LIN {X 0,Y 259.412,Z 737.757,A -85,B 0,C 180,E1 -19010.279,E2 -19010.279} C_VEL
LIN {X 0,Y 258.208,Z 750.679,A -85,B 0,C 180,E1 -19011.308,E2 -19011.308} C_VEL
LIN {X 0,Y 256.889,Z 762.034,A -85,B 0,C 180,E1 -19012.52,E2 -19012.52} C_VEL
LIN {X 0,Y 255.443,Z 772.557,A -85,B 0,C 180,E1 -19013.942,E2 -19013.942} C_VEL
LIN {X 0,Y 253.814,Z 782.677,A -85,B 0,C 180,E1 -19015.634,E2 -19015.634} C_VEL
LIN {X 0,Y 252.288,Z 792.086,A -85,B 0,C 180,E1 -19017.598,E2 -19017.598} C_VEL
LIN {X 0,Y 250.698,Z 801.193,A -85,B 0,C 180,E1 -19019.969,E2 -19019.969} C_VEL
LIN {X 0,Y 249.415,Z 808.562,A -85,B 0,C 180,E1 -19022.369,E2 -19022.369} C_VEL
LIN {X 0,Y 248.447,Z 814.636,A -85,B 0,C 180,E1 -19024.883,E2 -19024.883} C_VEL
LIN {X 0,Y 247.734,Z 819.375,A -85,B 0,C 180,E1 -19027.409,E2 -19027.409} C_VEL
LIN {X 0,Y 247.173,Z 822.833,A -85,B 0,C 180,E1 -19029.853,E2 -19029.853} C_VEL
LIN {X 0,Y 246.789,Z 825.879,A -85,B 0,C 180,E1 -19033.114,E2 -19033.114} C_VEL
LIN {X 0,Y 246.747,Z 826.996,A -85,B 0,C 180,E1 -19035.402,E2 -19035.402} C_VEL
LIN {X 0,Y 246.905,Z 827.33,A -85,B 0,C 180,E1 -19037.736,E2 -19037.736} C_VEL
LIN {X 0,Y 247.35,Z 826.83,A -85,B 0,C 180,E1 -19040.097,E2 -19040.097} C_VEL
LIN {X 0,Y 248.008,Z 825.441,A -85,B 0,C 180,E1 -19042.508,E2 -19042.508} C_VEL
LIN {X 0,Y 249.202,Z 822.178,A -85,B 0,C 180,E1 -19045.665,E2 -19045.665} C_VEL
LIN {X 0,Y 250.317,Z 819.07,A -85,B 0,C 180,E1 -19047.762,E2 -19047.762} C_VEL
LIN {X 0,Y 252.087,Z 813.878,A -85,B 0,C 180,E1 -19050.417,E2 -19050.417} C_VEL
LIN {X 0,Y 254.053,Z 807.904,A -85,B 0,C 180,E1 -19052.774,E2 -19052.774} C_VEL
LIN {X 0,Y 256.165,Z 801.239,A -85,B 0,C 180,E1 -19054.87,E2 -19054.87} C_VEL
LIN {X 0,Y 258.677,Z 792.614,A -85,B 0,C 180,E1 -19057.05,E2 -19057.05} C_VEL
LIN {X 0,Y 261.487,Z 782.053,A -85,B 0,C 180,E1 -19059.139,E2 -19059.139} C_VEL
LIN {X 0,Y 263.88,Z 771.777,A -85,B 0,C 180,E1 -19060.757,E2 -19060.757} C_VEL
LIN {X 0,Y 265.994,Z 761.633,A -85,B 0,C 180,E1 -19062.019,E2 -19062.019} C_VEL
LIN {X 0,Y 267.994,Z 749.161,A -85,B 0,C 180,E1 -19063.235,E2 -19063.235} C_VEL
LIN {X 0,Y 269.511,Z 735.967,A -85,B 0,C 180,E1 -19064.192,E2 -19064.192} C_VEL
LIN {X 0,Y 270.642,Z 723.077,A -85,B 0,C 180,E1 -19064.783,E2 -19064.783} C_VEL
LIN {X 0,Y 273.912,Z 663.749,A -85,B 0,C 180,E1 -19066.609,E2 -19066.609} C_VEL
LIN {X 0,Y 268.766,Z 652.292,A -85,B 0,C 180,E1 -19068.036,E2 -19068.036} C_VEL
LIN {X 0,Y 263.392,Z 642.224,A -85,B 0,C 180,E1 -19069.562,E2 -19069.562} C_VEL
LIN {X 0,Y 255.899,Z 629.943,A -85,B 0,C 180,E1 -19071.86,E2 -19071.86} C_VEL
LIN {X 0,Y 252.994,Z 625.595,A -85,B 0,C 180,E1 -19072.82,E2 -19072.82} C_VEL
LIN {X 0,Y 250.001,Z 621.447,A -85,B 0,C 180,E1 -19073.848,E2 -19073.848} C_VEL
LIN {X 0,Y 249.794,Z 620.987,A -85,B 0,C 180,E1 -19073.944,E2 -19073.944} C_VEL
LIN {X 0,Y 249.398,Z 619.817,A -85,B 0,C 180,E1 -19074.835,E2 -19074.835} C_VEL
LIN {X 0,Y 248.951,Z 619.475,A -85,B 0,C 180,E1 -19075.705,E2 -19075.705} C_VEL
LIN {X 0,Y 247.095,Z 619.707,A -85,B 0,C 180,E1 -19077.471,E2 -19077.471} C_VEL
LIN {X 0,Y 242.966,Z 620.26,A -85,B 0,C 180,E1 -19081.103,E2 -19081.103} C_VEL
LIN {X 0,Y 242.555,Z 620.265,A -85,B 0,C 180,E1 -19082.049,E2 -19082.049} C_VEL
LIN {X 0,Y 242.429,Z 620.281,A -85,B 0,C 180,E1 -19086.66,E2 -19086.66} C_VEL
LIN {X 0,Y 242.31,Z 620.295,A -85,B 0,C 180,E1 -19090.023,E2 -19090.023} C_VEL
LIN {X 0,Y 242.16,Z 620.316,A -85,B 0,C 180,E1 -19095.142,E2 -19095.142} C_VEL
LIN {X 0,Y 242.069,Z 620.326,A -85,B 0,C 180,E1 -19098.625,E2 -19098.625} C_VEL
LIN {X 0,Y 242.01,Z 620.331,A -85,B 0,C 180,E1 -19102.181,E2 -19102.181} C_VEL
LIN {X 0,Y 242.064,Z 620.322,A -85,B 0,C 180,E1 -19105.839,E2 -19105.839} C_VEL
LIN {X 0,Y 242.005,Z 620.33,A -85,B 0,C 180,E1 -19109.584,E2 -19109.584} C_VEL
LIN {X 0,Y 241.989,Z 620.338,A -85,B 0,C 180,E1 -19113.492,E2 -19113.492} C_VEL
LIN {X 0,Y 242.009,Z 620.332,A -85,B 0,C 180,E1 -19117.579,E2 -19117.579} C_VEL
LIN {X 0,Y 241.997,Z 620.472,A -85,B 0,C 180,E1 -19120.82,E2 -19120.82} C_VEL
LIN {X 0,Y 243.717,Z 626.064,A -85,B 0,C 180,E1 -19124.952,E2 -19124.952} C_VEL
LIN {X 0,Y 245.608,Z 632.24,A -85,B 0,C 180,E1 -19128.843,E2 -19128.843} C_VEL
LIN {X 0,Y 246.3,Z 634.523,A -85,B 0,C 180,E1 -19130.1,E2 -19130.1} C_VEL
LIN {X 0,Y 248.796,Z 639.028,A -85,B 0,C 180,E1 -19131.04,E2 -19131.04} C_VEL
LIN {X 0,Y 250.278,Z 641.401,A -85,B 0,C 180,E1 -19131.566,E2 -19131.566} C_VEL
LIN {X 0,Y 253.661,Z 647.375,A -85,B 0,C 180,E1 -19132.733,E2 -19132.733} C_VEL
LIN {X 0,Y 258.381,Z 656.509,A -85,B 0,C 180,E1 -19134.278,E2 -19134.278} C_VEL
LIN {X 0,Y 263.504,Z 667.81,A -85,B 0,C 180,E1 -19135.875,E2 -19135.875} C_VEL
LIN {X 0,Y 264.479,Z 670.795,A -85,B 0,C 180,E1 -19136.199,E2 -19136.199} C_VEL
LIN {X 0,Y 266.594,Z 687.408,A -85,B 0,C 180,E1 -19137.319,E2 -19137.319} C_VEL
LIN {X 0,Y 267.059,Z 694.958,A -85,B 0,C 180,E1 -19137.724,E2 -19137.724} C_VEL
LIN {X 0,Y 264.07,Z 745.91,A -85,B 0,C 180,E1 -19139.343,E2 -19139.343} C_VEL
LIN {X 0,Y 262.439,Z 760.152,A -85,B 0,C 180,E1 -19140.082,E2 -19140.082} C_VEL
LIN {X 0,Y 260.483,Z 771.827,A -85,B 0,C 180,E1 -19140.946,E2 -19140.946} C_VEL
LIN {X 0,Y 257.997,Z 784.148,A -85,B 0,C 180,E1 -19142.194,E2 -19142.194} C_VEL
LIN {X 0,Y 255.328,Z 795.293,A -85,B 0,C 180,E1 -19143.651,E2 -19143.651} C_VEL
LIN {X 0,Y 252.655,Z 805.45,A -85,B 0,C 180,E1 -19145.34,E2 -19145.34} C_VEL
LIN {X 0,Y 249.936,Z 814.673,A -85,B 0,C 180,E1 -19147.255,E2 -19147.255} C_VEL
LIN {X 0,Y 247.165,Z 823.89,A -85,B 0,C 180,E1 -19149.66,E2 -19149.66} C_VEL
LIN {X 0,Y 244.913,Z 831.116,A -85,B 0,C 180,E1 -19152.033,E2 -19152.033} C_VEL
LIN {X 0,Y 243.367,Z 836.122,A -85,B 0,C 180,E1 -19154.078,E2 -19154.078} C_VEL
LIN {X 0,Y 241.756,Z 841.03,A -85,B 0,C 180,E1 -19156.552,E2 -19156.552} C_VEL
LIN {X 0,Y 240.801,Z 844.831,A -85,B 0,C 180,E1 -19159.065,E2 -19159.065} C_VEL
LIN {X 0,Y 240.187,Z 847.629,A -85,B 0,C 180,E1 -19161.587,E2 -19161.587} C_VEL
LIN {X 0,Y 239.985,Z 848.983,A -85,B 0,C 180,E1 -19163.273,E2 -19163.273} C_VEL
LIN {X 0,Y 239.883,Z 849.917,A -85,B 0,C 180,E1 -19164.958,E2 -19164.958} C_VEL
LIN {X 0,Y 239.923,Z 850.416,A -85,B 0,C 180,E1 -19166.641,E2 -19166.641} C_VEL
LIN {X 0,Y 239.986,Z 850.517,A -85,B 0,C 180,E1 -19168.322,E2 -19168.322} C_VEL
LIN {X 0,Y 240.04,Z 850.216,A -85,B 0,C 180,E1 -19170,E2 -19170} C_VEL
LIN {X 0,Y 240.008,Z 849.483,A -85,B 0,C 180,E1 -19171.678,E2 -19171.678} C_VEL
LIN {X 0,Y 239.972,Z 848.286,A -85,B 0,C 180,E1 -19173.358,E2 -19173.358} C_VEL
LIN {X 0,Y 239.954,Z 846.459,A -85,B 0,C 180,E1 -19175.23,E2 -19175.23} C_VEL
LIN {X 0,Y 240.119,Z 843.345,A -85,B 0,C 180,E1 -19177.568,E2 -19177.568} C_VEL
LIN {X 0,Y 240.537,Z 838.897,A -85,B 0,C 180,E1 -19180.096,E2 -19180.096} C_VEL
LIN {X 0,Y 241.246,Z 833.19,A -85,B 0,C 180,E1 -19182.62,E2 -19182.62} C_VEL
LIN {X 0,Y 242.509,Z 826.029,A -85,B 0,C 180,E1 -19185.119,E2 -19185.119} C_VEL
LIN {X 0,Y 243.903,Z 817.46,A -85,B 0,C 180,E1 -19187.495,E2 -19187.495} C_VEL
LIN {X 0,Y 245.216,Z 809.762,A -85,B 0,C 180,E1 -19189.243,E2 -19189.243} C_VEL
LIN {X 0,Y 247.061,Z 798.798,A -85,B 0,C 180,E1 -19191.265,E2 -19191.265} C_VEL
LIN {X 0,Y 248.915,Z 787.83,A -85,B 0,C 180,E1 -19192.844,E2 -19192.844} C_VEL
LIN {X 0,Y 250.596,Z 775.59,A -85,B 0,C 180,E1 -19194.214,E2 -19194.214} C_VEL
LIN {X 0,Y 252.105,Z 762.896,A -85,B 0,C 180,E1 -19195.268,E2 -19195.268} C_VEL
LIN {X 0,Y 253.179,Z 749.404,A -85,B 0,C 180,E1 -19196.036,E2 -19196.036} C_VEL
LIN {X 0,Y 254.298,Z 723.087,A -85,B 0,C 180,E1 -19196.916,E2 -19196.916} C_VEL
LIN {X 0,Y 255.425,Z 690.334,A -85,B 0,C 180,E1 -19197.95,E2 -19197.95} C_VEL
LIN {X 0,Y 250.396,Z 651.358,A -85,B 0,C 180,E1 -19199.786,E2 -19199.786} C_VEL
LIN {X 0,Y 245.876,Z 638.506,A -85,B 0,C 180,E1 -19200.761,E2 -19200.761} C_VEL
LIN {X 0,Y 243.435,Z 626.587,A -85,B 0,C 180,E1 -19205.267,E2 -19205.267} C_VEL
LIN {X 0,Y 242.027,Z 620.336,A -85,B 0,C 180,E1 -19207.771,E2 -19207.771} C_VEL
LIN {X 0,Y 241.968,Z 620.346,A -85,B 0,C 180,E1 -19211.915,E2 -19211.915} C_VEL
LIN {X 0,Y 241.977,Z 620.345,A -85,B 0,C 180,E1 -19216.559,E2 -19216.559} C_VEL
LIN {X 0,Y 241.987,Z 620.342,A -85,B 0,C 180,E1 -19220.286,E2 -19220.286} C_VEL
LIN {X 0,Y 242.035,Z 620.337,A -85,B 0,C 180,E1 -19224.496,E2 -19224.496} C_VEL
LIN {X 0,Y 241.974,Z 620.343,A -85,B 0,C 180,E1 -19228.479,E2 -19228.479} C_VEL
LIN {X 0,Y 242.004,Z 620.338,A -85,B 0,C 180,E1 -19232.311,E2 -19232.311} C_VEL
LIN {X 0,Y 242.037,Z 620.333,A -85,B 0,C 180,E1 -19236.013,E2 -19236.013} C_VEL
LIN {X 0,Y 242.031,Z 620.334,A -85,B 0,C 180,E1 -19239.607,E2 -19239.607} C_VEL
LIN {X 0,Y 242.16,Z 620.32,A -85,B 0,C 180,E1 -19243.277,E2 -19243.277} C_VEL
LIN {X 0,Y 242.181,Z 620.314,A -85,B 0,C 180,E1 -19248.279,E2 -19248.279} C_VEL
LIN {X 0,Y 242.421,Z 620.284,A -85,B 0,C 180,E1 -19251.665,E2 -19251.665} C_VEL
LIN {X 0,Y 242.255,Z 620.308,A -85,B 0,C 180,E1 -19255.006,E2 -19255.006} C_VEL
LIN {X 0,Y 242.631,Z 620.257,A -85,B 0,C 180,E1 -19258.339,E2 -19258.339} C_VEL
LIN {X 0,Y 242.631,Z 620.254,A -85,B 0,C 180,E1 -19261.659,E2 -19261.659} C_VEL
LIN {X 0,Y 242.423,Z 620.285,A -85,B 0,C 180,E1 -19266.702,E2 -19266.702} C_VEL
LIN {X 0,Y 242.308,Z 620.297,A -85,B 0,C 180,E1 -19270.021,E2 -19270.021} C_VEL
LIN {X 0,Y 242.15,Z 620.313,A -85,B 0,C 180,E1 -19275.141,E2 -19275.141} C_VEL
LIN {X 0,Y 242.064,Z 620.329,A -85,B 0,C 180,E1 -19278.624,E2 -19278.624} C_VEL
LIN {X 0,Y 242.007,Z 620.334,A -85,B 0,C 180,E1 -19282.18,E2 -19282.18} C_VEL
LIN {X 0,Y 242.061,Z 620.322,A -85,B 0,C 180,E1 -19285.838,E2 -19285.838} C_VEL
LIN {X 0,Y 242.001,Z 620.336,A -85,B 0,C 180,E1 -19289.583,E2 -19289.583} C_VEL
LIN {X 0,Y 241.986,Z 620.339,A -85,B 0,C 180,E1 -19293.491,E2 -19293.491} C_VEL
LIN {X 0,Y 242.007,Z 620.329,A -85,B 0,C 180,E1 -19297.578,E2 -19297.578} C_VEL
LIN {X 0,Y 241.979,Z 620.341,A -85,B 0,C 180,E1 -19301.912,E2 -19301.912} C_VEL
LIN {X 0,Y 241.981,Z 620.34,A -85,B 0,C 180,E1 -19306.558,E2 -19306.558} C_VEL
LIN {X 0,Y 241.977,Z 620.335,A -85,B 0,C 180,E1 -19310.286,E2 -19310.286} C_VEL
LIN {X 0,Y 242.032,Z 620.338,A -85,B 0,C 180,E1 -19314.498,E2 -19314.498} C_VEL
LIN {X 0,Y 241.97,Z 620.339,A -85,B 0,C 180,E1 -19318.48,E2 -19318.48} C_VEL
LIN {X 0,Y 241.998,Z 620.339,A -85,B 0,C 180,E1 -19322.312,E2 -19322.312} C_VEL
LIN {X 0,Y 242.053,Z 620.331,A -85,B 0,C 180,E1 -19326.016,E2 -19326.016} C_VEL
LIN {X 0,Y 242.034,Z 620.333,A -85,B 0,C 180,E1 -19329.608,E2 -19329.608} C_VEL
LIN {X 0,Y 242.16,Z 620.318,A -85,B 0,C 180,E1 -19333.278,E2 -19333.278} C_VEL
LIN {X 0,Y 242.184,Z 620.315,A -85,B 0,C 180,E1 -19338.28,E2 -19338.28} C_VEL
LIN {X 0,Y 242.423,Z 620.283,A -85,B 0,C 180,E1 -19341.666,E2 -19341.666} C_VEL
LIN {X 0,Y 242.257,Z 620.307,A -85,B 0,C 180,E1 -19345.007,E2 -19345.007} C_VEL
LIN {X 0,Y 242.634,Z 620.258,A -85,B 0,C 180,E1 -19348.34,E2 -19348.34} C_VEL
LIN {X 0,Y 242.634,Z 620.259,A -85,B 0,C 180,E1 -19351.66,E2 -19351.66} C_VEL
LIN {X 0,Y 242.421,Z 620.287,A -85,B 0,C 180,E1 -19356.659,E2 -19356.659} C_VEL
LIN {X 0,Y 242.264,Z 620.307,A -85,B 0,C 180,E1 -19360.024,E2 -19360.024} C_VEL
LIN {X 0,Y 242.179,Z 620.32,A -85,B 0,C 180,E1 -19364.119,E2 -19364.119} C_VEL
LIN {X 0,Y 243.197,Z 623.213,A -85,B 0,C 180,E1 -19364.353,E2 -19364.353} C_VEL
LIN {X 0,Y 250.975,Z 640.87,A -85,B 0,C 180,E1 -19365.802,E2 -19365.802} C_VEL
LIN {X 0,Y 256.337,Z 655.837,A -85,B 0,C 180,E1 -19366.839,E2 -19366.839} C_VEL
LIN {X 0,Y 253.594,Z 724.318,A -85,B 0,C 180,E1 -19369.008,E2 -19369.008} C_VEL
LIN {X 0,Y 252.699,Z 738.217,A -85,B 0,C 180,E1 -19369.786,E2 -19369.786} C_VEL
LIN {X 0,Y 251.52,Z 750.319,A -85,B 0,C 180,E1 -19370.763,E2 -19370.763} C_VEL
LIN {X 0,Y 249.946,Z 763.385,A -85,B 0,C 180,E1 -19372.202,E2 -19372.202} C_VEL
LIN {X 0,Y 248.319,Z 774.48,A -85,B 0,C 180,E1 -19373.774,E2 -19373.774} C_VEL
LIN {X 0,Y 246.509,Z 785.512,A -85,B 0,C 180,E1 -19375.771,E2 -19375.771} C_VEL
LIN {X 0,Y 244.819,Z 795.48,A -85,B 0,C 180,E1 -19378.037,E2 -19378.037} C_VEL
LIN {X 0,Y 243.527,Z 802.572,A -85,B 0,C 180,E1 -19380.03,E2 -19380.03} C_VEL
LIN {X 0,Y 242.184,Z 810.192,A -85,B 0,C 180,E1 -19382.697,E2 -19382.697} C_VEL
LIN {X 0,Y 241.131,Z 816.741,A -85,B 0,C 180,E1 -19385.655,E2 -19385.655} C_VEL
LIN {X 0,Y 240.498,Z 820.552,A -85,B 0,C 180,E1 -19387.908,E2 -19387.908} C_VEL
LIN {X 0,Y 239.986,Z 823.774,A -85,B 0,C 180,E1 -19390.413,E2 -19390.413} C_VEL
LIN {X 0,Y 239.704,Z 825.962,A -85,B 0,C 180,E1 -19392.864,E2 -19392.864} C_VEL
LIN {X 0,Y 239.65,Z 827.245,A -85,B 0,C 180,E1 -19395.267,E2 -19395.267} C_VEL
LIN {X 0,Y 239.802,Z 827.71,A -85,B 0,C 180,E1 -19397.619,E2 -19397.619} C_VEL
LIN {X 0,Y 240.228,Z 827.369,A -85,B 0,C 180,E1 -19399.939,E2 -19399.939} C_VEL
LIN {X 0,Y 240.817,Z 826.278,A -85,B 0,C 180,E1 -19402.204,E2 -19402.204} C_VEL
LIN {X 0,Y 242.079,Z 823.294,A -85,B 0,C 180,E1 -19405.568,E2 -19405.568} C_VEL
LIN {X 0,Y 243.825,Z 818.733,A -85,B 0,C 180,E1 -19408.747,E2 -19408.747} C_VEL
LIN {X 0,Y 245.899,Z 813.054,A -85,B 0,C 180,E1 -19411.589,E2 -19411.589} C_VEL
LIN {X 0,Y 248.423,Z 805.642,A -85,B 0,C 180,E1 -19414.361,E2 -19414.361} C_VEL
LIN {X 0,Y 250.798,Z 798.49,A -85,B 0,C 180,E1 -19416.465,E2 -19416.465} C_VEL
LIN {X 0,Y 253.583,Z 789.189,A -85,B 0,C 180,E1 -19418.67,E2 -19418.67} C_VEL
LIN {X 0,Y 256.377,Z 778.677,A -85,B 0,C 180,E1 -19420.619,E2 -19420.619} C_VEL
LIN {X 0,Y 258.893,Z 767.889,A -85,B 0,C 180,E1 -19422.2,E2 -19422.2} C_VEL
LIN {X 0,Y 261.273,Z 755.768,A -85,B 0,C 180,E1 -19423.565,E2 -19423.565} C_VEL
LIN {X 0,Y 263.136,Z 743.169,A -85,B 0,C 180,E1 -19424.642,E2 -19424.642} C_VEL
LIN {X 0,Y 264.315,Z 731.972,A -85,B 0,C 180,E1 -19425.345,E2 -19425.345} C_VEL
LIN {X 0,Y 265.338,Z 718.751,A -85,B 0,C 180,E1 -19425.868,E2 -19425.868} C_VEL
LIN {X 0,Y 268.479,Z 666.273,A -85,B 0,C 180,E1 -19427.495,E2 -19427.495} C_VEL
LIN {X 0,Y 263.835,Z 655.832,A -85,B 0,C 180,E1 -19428.859,E2 -19428.859} C_VEL
LIN {X 0,Y 258.895,Z 646.535,A -85,B 0,C 180,E1 -19430.35,E2 -19430.35} C_VEL
LIN {X 0,Y 252.272,Z 635.35,A -85,B 0,C 180,E1 -19432.497,E2 -19432.497} C_VEL
LIN {X 0,Y 248.99,Z 630.59,A -85,B 0,C 180,E1 -19433.63,E2 -19433.63} C_VEL
LIN {X 0,Y 245.83,Z 626.212,A -85,B 0,C 180,E1 -19434.773,E2 -19434.773} C_VEL
LIN {X 0,Y 243.118,Z 622.829,A -85,B 0,C 180,E1 -19435.805,E2 -19435.805} C_VEL
LIN {X 0,Y 242.633,Z 621.629,A -85,B 0,C 180,E1 -19436.056,E2 -19436.056} C_VEL
LIN {X 0,Y 242.455,Z 620.283,A -85,B 0,C 180,E1 -19437.197,E2 -19437.197} C_VEL
LIN {X 0,Y 242.693,Z 620.256,A -85,B 0,C 180,E1 -19440.001,E2 -19440.001} C_VEL
LIN {X 0,Y 242.555,Z 620.265,A -85,B 0,C 180,E1 -19442.049,E2 -19442.049} C_VEL
LIN {X 0,Y 241.713,Z 620.372,A -85,B 0,C 180,E1 -19443.434,E2 -19443.434} C_VEL
LIN {X 0,Y 238.808,Z 620.738,A -85,B 0,C 180,E1 -19445.695,E2 -19445.695} C_VEL
LIN {X 0,Y 236.434,Z 621.032,A -85,B 0,C 180,E1 -19447.537,E2 -19447.537} C_VEL
LIN {X 0,Y 235.407,Z 621.159,A -85,B 0,C 180,E1 -19448.965,E2 -19448.965} C_VEL
LIN {X 0,Y 235.312,Z 621.167,A -85,B 0,C 180,E1 -19449.449,E2 -19449.449} C_VEL
LIN {X 0,Y 235.1,Z 621.197,A -85,B 0,C 180,E1 -19453.837,E2 -19453.837} C_VEL
LIN {X 0,Y 235.065,Z 621.204,A -85,B 0,C 180,E1 -19457.397,E2 -19457.397} C_VEL
LIN {X 0,Y 234.99,Z 621.206,A -85,B 0,C 180,E1 -19462.011,E2 -19462.011} C_VEL
LIN {X 0,Y 234.965,Z 621.209,A -85,B 0,C 180,E1 -19466.659,E2 -19466.659} C_VEL
LIN {X 0,Y 234.921,Z 621.219,A -85,B 0,C 180,E1 -19470.57,E2 -19470.57} C_VEL
LIN {X 0,Y 234.959,Z 621.208,A -85,B 0,C 180,E1 -19474.634,E2 -19474.634} C_VEL
LIN {X 0,Y 235.001,Z 621.287,A -85,B 0,C 180,E1 -19478.358,E2 -19478.358} C_VEL
LIN {X 0,Y 236.76,Z 626.908,A -85,B 0,C 180,E1 -19483.059,E2 -19483.059} C_VEL
LIN {X 0,Y 238.792,Z 633.746,A -85,B 0,C 180,E1 -19487.726,E2 -19487.726} C_VEL
LIN {X 0,Y 241.533,Z 638.403,A -85,B 0,C 180,E1 -19488.894,E2 -19488.894} C_VEL
LIN {X 0,Y 243.004,Z 640.499,A -85,B 0,C 180,E1 -19489.472,E2 -19489.472} C_VEL
LIN {X 0,Y 246.93,Z 647.301,A -85,B 0,C 180,E1 -19490.978,E2 -19490.978} C_VEL
LIN {X 0,Y 249.888,Z 652.716,A -85,B 0,C 180,E1 -19492.061,E2 -19492.061} C_VEL
LIN {X 0,Y 254.084,Z 660.972,A -85,B 0,C 180,E1 -19493.507,E2 -19493.507} C_VEL
LIN {X 0,Y 258.76,Z 671.596,A -85,B 0,C 180,E1 -19495.067,E2 -19495.067} C_VEL
LIN {X 0,Y 259.488,Z 674.129,A -85,B 0,C 180,E1 -19495.337,E2 -19495.337} C_VEL
LIN {X 0,Y 261.522,Z 691.303,A -85,B 0,C 180,E1 -19496.509,E2 -19496.509} C_VEL
LIN {X 0,Y 261.642,Z 696.477,A -85,B 0,C 180,E1 -19496.758,E2 -19496.758} C_VEL
LIN {X 0,Y 258.552,Z 745.528,A -85,B 0,C 180,E1 -19498.354,E2 -19498.354} C_VEL
LIN {X 0,Y 256.886,Z 759.375,A -85,B 0,C 180,E1 -19499.082,E2 -19499.082} C_VEL
LIN {X 0,Y 254.753,Z 771.597,A -85,B 0,C 180,E1 -19499.999,E2 -19499.999} C_VEL
LIN {X 0,Y 252.179,Z 783.881,A -85,B 0,C 180,E1 -19501.267,E2 -19501.267} C_VEL
LIN {X 0,Y 249.375,Z 795.014,A -85,B 0,C 180,E1 -19502.745,E2 -19502.745} C_VEL
LIN {X 0,Y 246.539,Z 805.158,A -85,B 0,C 180,E1 -19504.459,E2 -19504.459} C_VEL
LIN {X 0,Y 243.426,Z 815.185,A -85,B 0,C 180,E1 -19506.611,E2 -19506.611} C_VEL
LIN {X 0,Y 240.552,Z 824.083,A -85,B 0,C 180,E1 -19509.029,E2 -19509.029} C_VEL
LIN {X 0,Y 238.149,Z 831.268,A -85,B 0,C 180,E1 -19511.504,E2 -19511.504} C_VEL
LIN {X 0,Y 236.538,Z 836.205,A -85,B 0,C 180,E1 -19513.605,E2 -19513.605} C_VEL
LIN {X 0,Y 234.827,Z 841.024,A -85,B 0,C 180,E1 -19516.148,E2 -19516.148} C_VEL
LIN {X 0,Y 233.8,Z 844.738,A -85,B 0,C 180,E1 -19518.733,E2 -19518.733} C_VEL
LIN {X 0,Y 233.129,Z 847.449,A -85,B 0,C 180,E1 -19521.331,E2 -19521.331} C_VEL
LIN {X 0,Y 232.91,Z 848.756,A -85,B 0,C 180,E1 -19523.068,E2 -19523.068} C_VEL
LIN {X 0,Y 232.803,Z 849.694,A -85,B 0,C 180,E1 -19525.029,E2 -19525.029} C_VEL
LIN {X 0,Y 232.914,Z 850.149,A -85,B 0,C 180,E1 -19528.271,E2 -19528.271} C_VEL
LIN {X 0,Y 232.967,Z 849.81,A -85,B 0,C 180,E1 -19530,E2 -19530} C_VEL
LIN {X 0,Y 232.937,Z 849.007,A -85,B 0,C 180,E1 -19531.729,E2 -19531.729} C_VEL
LIN {X 0,Y 232.887,Z 847.771,A -85,B 0,C 180,E1 -19533.46,E2 -19533.46} C_VEL
LIN {X 0,Y 232.903,Z 845.082,A -85,B 0,C 180,E1 -19536.062,E2 -19536.062} C_VEL
LIN {X 0,Y 233.177,Z 841.314,A -85,B 0,C 180,E1 -19538.667,E2 -19538.667} C_VEL
LIN {X 0,Y 233.735,Z 836.362,A -85,B 0,C 180,E1 -19541.27,E2 -19541.27} C_VEL
LIN {X 0,Y 234.672,Z 830.083,A -85,B 0,C 180,E1 -19543.862,E2 -19543.862} C_VEL
LIN {X 0,Y 236.043,Z 822.224,A -85,B 0,C 180,E1 -19546.43,E2 -19546.43} C_VEL
LIN {X 0,Y 236.942,Z 816.796,A -85,B 0,C 180,E1 -19547.9,E2 -19547.9} C_VEL
LIN {X 0,Y 238.858,Z 806.46,A -85,B 0,C 180,E1 -19550.225,E2 -19550.225} C_VEL
LIN {X 0,Y 240.464,Z 797.275,A -85,B 0,C 180,E1 -19551.878,E2 -19551.878} C_VEL
LIN {X 0,Y 242.315,Z 785.977,A -85,B 0,C 180,E1 -19553.502,E2 -19553.502} C_VEL
LIN {X 0,Y 243.835,Z 775.346,A -85,B 0,C 180,E1 -19554.703,E2 -19554.703} C_VEL
LIN {X 0,Y 245.37,Z 762.692,A -85,B 0,C 180,E1 -19555.785,E2 -19555.785} C_VEL
LIN {X 0,Y 246.493,Z 749.289,A -85,B 0,C 180,E1 -19556.569,E2 -19556.569} C_VEL
LIN {X 0,Y 247.58,Z 724.665,A -85,B 0,C 180,E1 -19557.421,E2 -19557.421} C_VEL
LIN {X 0,Y 248.733,Z 690.762,A -85,B 0,C 180,E1 -19558.527,E2 -19558.527} C_VEL
LIN {X 0,Y 243.985,Z 653.427,A -85,B 0,C 180,E1 -19560.349,E2 -19560.349} C_VEL
LIN {X 0,Y 238.628,Z 638.243,A -85,B 0,C 180,E1 -19561.518,E2 -19561.518} C_VEL
LIN {X 0,Y 236.148,Z 626.33,A -85,B 0,C 180,E1 -19566.192,E2 -19566.192} C_VEL
LIN {X 0,Y 234.976,Z 621.217,A -85,B 0,C 180,E1 -19568.36,E2 -19568.36} C_VEL
LIN {X 0,Y 234.957,Z 621.219,A -85,B 0,C 180,E1 -19573.468,E2 -19573.468} C_VEL
LIN {X 0,Y 234.952,Z 621.22,A -85,B 0,C 180,E1 -19576.528,E2 -19576.528} C_VEL
LIN {X 0,Y 234.954,Z 621.218,A -85,B 0,C 180,E1 -19581.085,E2 -19581.085} C_VEL
LIN {X 0,Y 234.959,Z 621.217,A -85,B 0,C 180,E1 -19585.366,E2 -19585.366} C_VEL
LIN {X 0,Y 234.967,Z 621.214,A -85,B 0,C 180,E1 -19590.156,E2 -19590.156} C_VEL
LIN {X 0,Y 234.991,Z 621.208,A -85,B 0,C 180,E1 -19593.793,E2 -19593.793} C_VEL
LIN {X 0,Y 234.994,Z 621.215,A -85,B 0,C 180,E1 -19598.967,E2 -19598.967} C_VEL
LIN {X 0,Y 235.092,Z 621.198,A -85,B 0,C 180,E1 -19603.059,E2 -19603.059} C_VEL
LIN {X 0,Y 235.113,Z 621.195,A -85,B 0,C 180,E1 -19607.921,E2 -19607.921} C_VEL
LIN {X 0,Y 235.371,Z 621.161,A -85,B 0,C 180,E1 -19611.413,E2 -19611.413} C_VEL
LIN {X 0,Y 235.397,Z 621.16,A -85,B 0,C 180,E1 -19613.14,E2 -19613.14} C_VEL
LIN {X 0,Y 235.591,Z 621.134,A -85,B 0,C 180,E1 -19618.29,E2 -19618.29} C_VEL
LIN {X 0,Y 235.591,Z 621.13,A -85,B 0,C 180,E1 -19621.709,E2 -19621.709} C_VEL
LIN {X 0,Y 235.397,Z 621.161,A -85,B 0,C 180,E1 -19626.858,E2 -19626.858} C_VEL
LIN {X 0,Y 235.232,Z 621.177,A -85,B 0,C 180,E1 -19630.326,E2 -19630.326} C_VEL
LIN {X 0,Y 235.101,Z 621.193,A -85,B 0,C 180,E1 -19635.606,E2 -19635.606} C_VEL
LIN {X 0,Y 235.001,Z 621.209,A -85,B 0,C 180,E1 -19639.205,E2 -19639.205} C_VEL
LIN {X 0,Y 234.955,Z 621.21,A -85,B 0,C 180,E1 -19642.882,E2 -19642.882} C_VEL
LIN {X 0,Y 234.962,Z 621.206,A -85,B 0,C 180,E1 -19646.657,E2 -19646.657} C_VEL
LIN {X 0,Y 234.917,Z 621.22,A -85,B 0,C 180,E1 -19650.569,E2 -19650.569} C_VEL
LIN {X 0,Y 234.955,Z 621.212,A -85,B 0,C 180,E1 -19654.633,E2 -19654.633} C_VEL
LIN {X 0,Y 234.961,Z 621.207,A -85,B 0,C 180,E1 -19658.952,E2 -19658.952} C_VEL
LIN {X 0,Y 234.96,Z 621.215,A -85,B 0,C 180,E1 -19663.468,E2 -19663.468} C_VEL
LIN {X 0,Y 234.956,Z 621.215,A -85,B 0,C 180,E1 -19666.531,E2 -19666.531} C_VEL
LIN {X 0,Y 234.95,Z 621.213,A -85,B 0,C 180,E1 -19671.086,E2 -19671.086} C_VEL
LIN {X 0,Y 234.956,Z 621.216,A -85,B 0,C 180,E1 -19675.367,E2 -19675.367} C_VEL
LIN {X 0,Y 234.918,Z 621.213,A -85,B 0,C 180,E1 -19679.431,E2 -19679.431} C_VEL
LIN {X 0,Y 234.99,Z 621.212,A -85,B 0,C 180,E1 -19683.794,E2 -19683.794} C_VEL
LIN {X 0,Y 235.008,Z 621.211,A -85,B 0,C 180,E1 -19688.97,E2 -19688.97} C_VEL
LIN {X 0,Y 235.093,Z 621.2,A -85,B 0,C 180,E1 -19693.059,E2 -19693.059} C_VEL
LIN {X 0,Y 235.144,Z 621.191,A -85,B 0,C 180,E1 -19697.924,E2 -19697.924} C_VEL
LIN {X 0,Y 235.373,Z 621.162,A -85,B 0,C 180,E1 -19701.414,E2 -19701.414} C_VEL
LIN {X 0,Y 235.4,Z 621.161,A -85,B 0,C 180,E1 -19703.141,E2 -19703.141} C_VEL
LIN {X 0,Y 235.594,Z 621.135,A -85,B 0,C 180,E1 -19708.291,E2 -19708.291} C_VEL
LIN {X 0,Y 235.594,Z 621.136,A -85,B 0,C 180,E1 -19711.709,E2 -19711.709} C_VEL
LIN {X 0,Y 235.39,Z 621.164,A -85,B 0,C 180,E1 -19716.859,E2 -19716.859} C_VEL
LIN {X 0,Y 235.211,Z 621.185,A -85,B 0,C 180,E1 -19720.327,E2 -19720.327} C_VEL
LIN {X 0,Y 235.161,Z 621.324,A -85,B 0,C 180,E1 -19723.392,E2 -19723.392} C_VEL
LIN {X 0,Y 236.141,Z 624.059,A -85,B 0,C 180,E1 -19723.609,E2 -19723.609} C_VEL
LIN {X 0,Y 244.656,Z 643.104,A -85,B 0,C 180,E1 -19725.244,E2 -19725.244} C_VEL
LIN {X 0,Y 249.8,Z 657.943,A -85,B 0,C 180,E1 -19726.297,E2 -19726.297} C_VEL
LIN {X 0,Y 246.908,Z 724.994,A -85,B 0,C 180,E1 -19728.477,E2 -19728.477} C_VEL
LIN {X 0,Y 245.963,Z 738.863,A -85,B 0,C 180,E1 -19729.279,E2 -19729.279} C_VEL
LIN {X 0,Y 244.642,Z 751.869,A -85,B 0,C 180,E1 -19730.384,E2 -19730.384} C_VEL
LIN {X 0,Y 243.038,Z 764.664,A -85,B 0,C 180,E1 -19731.858,E2 -19731.858} C_VEL
LIN {X 0,Y 241.248,Z 776.1,A -85,B 0,C 180,E1 -19733.567,E2 -19733.567} C_VEL
LIN {X 0,Y 239.627,Z 785.71,A -85,B 0,C 180,E1 -19735.37,E2 -19735.37} C_VEL
LIN {X 0,Y 237.942,Z 795.373,A -85,B 0,C 180,E1 -19737.615,E2 -19737.615} C_VEL
LIN {X 0,Y 236.505,Z 803.084,A -85,B 0,C 180,E1 -19739.832,E2 -19739.832} C_VEL
LIN {X 0,Y 235.146,Z 810.594,A -85,B 0,C 180,E1 -19742.545,E2 -19742.545} C_VEL
LIN {X 0,Y 234.15,Z 816.516,A -85,B 0,C 180,E1 -19745.271,E2 -19745.271} C_VEL
LIN {X 0,Y 233.449,Z 820.627,A -85,B 0,C 180,E1 -19747.702,E2 -19747.702} C_VEL
LIN {X 0,Y 233.066,Z 822.793,A -85,B 0,C 180,E1 -19749.289,E2 -19749.289} C_VEL
LIN {X 0,Y 232.727,Z 825.249,A -85,B 0,C 180,E1 -19751.632,E2 -19751.632} C_VEL
LIN {X 0,Y 232.564,Z 826.959,A -85,B 0,C 180,E1 -19754.03,E2 -19754.03} C_VEL
LIN {X 0,Y 232.607,Z 827.905,A -85,B 0,C 180,E1 -19756.479,E2 -19756.479} C_VEL
LIN {X 0,Y 232.924,Z 828.02,A -85,B 0,C 180,E1 -19758.965,E2 -19758.965} C_VEL
LIN {X 0,Y 233.515,Z 827.27,A -85,B 0,C 180,E1 -19761.489,E2 -19761.489} C_VEL
LIN {X 0,Y 234.344,Z 825.614,A -85,B 0,C 180,E1 -19764.068,E2 -19764.068} C_VEL
LIN {X 0,Y 235.523,Z 822.97,A -85,B 0,C 180,E1 -19766.668,E2 -19766.668} C_VEL
LIN {X 0,Y 237.404,Z 818.392,A -85,B 0,C 180,E1 -19769.785,E2 -19769.785} C_VEL
LIN {X 0,Y 239.478,Z 812.979,A -85,B 0,C 180,E1 -19772.471,E2 -19772.471} C_VEL
LIN {X 0,Y 242.287,Z 805.43,A -85,B 0,C 180,E1 -19775.32,E2 -19775.32} C_VEL
LIN {X 0,Y 244.941,Z 797.696,A -85,B 0,C 180,E1 -19777.601,E2 -19777.601} C_VEL
LIN {X 0,Y 247.772,Z 788.647,A -85,B 0,C 180,E1 -19779.713,E2 -19779.713} C_VEL
LIN {X 0,Y 250.599,Z 778.442,A -85,B 0,C 180,E1 -19781.61,E2 -19781.61} C_VEL
LIN {X 0,Y 252.941,Z 768.831,A -85,B 0,C 180,E1 -19783.039,E2 -19783.039} C_VEL
LIN {X 0,Y 255.382,Z 757.256,A -85,B 0,C 180,E1 -19784.399,E2 -19784.399} C_VEL
LIN {X 0,Y 257.381,Z 744.94,A -85,B 0,C 180,E1 -19785.497,E2 -19785.497} C_VEL
LIN {X 0,Y 258.752,Z 733.037,A -85,B 0,C 180,E1 -19786.283,E2 -19786.283} C_VEL
LIN {X 0,Y 259.848,Z 720.243,A -85,B 0,C 180,E1 -19786.818,E2 -19786.818} C_VEL
LIN {X 0,Y 262.976,Z 668.382,A -85,B 0,C 180,E1 -19788.478,E2 -19788.478} C_VEL
LIN {X 0,Y 258.153,Z 657.637,A -85,B 0,C 180,E1 -19789.992,E2 -19789.992} C_VEL
LIN {X 0,Y 252.825,Z 647.884,A -85,B 0,C 180,E1 -19791.711,E2 -19791.711} C_VEL
LIN {X 0,Y 247.761,Z 639.457,A -85,B 0,C 180,E1 -19793.486,E2 -19793.486} C_VEL
LIN {X 0,Y 245.515,Z 636.084,A -85,B 0,C 180,E1 -19794.3,E2 -19794.3} C_VEL
LIN {X 0,Y 242.439,Z 631.782,A -85,B 0,C 180,E1 -19795.481,E2 -19795.481} C_VEL
LIN {X 0,Y 239.589,Z 627.891,A -85,B 0,C 180,E1 -19796.638,E2 -19796.638} C_VEL
LIN {X 0,Y 236.184,Z 623.303,A -85,B 0,C 180,E1 -19798.136,E2 -19798.136} C_VEL
LIN {X 0,Y 235.829,Z 622.264,A -85,B 0,C 180,E1 -19798.4,E2 -19798.4} C_VEL
LIN {X 0,Y 235.633,Z 621.132,A -85,B 0,C 180,E1 -19799.574,E2 -19799.574} C_VEL
LIN {X 0,Y 235.538,Z 621.14,A -85,B 0,C 180,E1 -19801.965,E2 -19801.965} C_VEL
LIN {X 0,Y 235.4,Z 621.156,A -85,B 0,C 180,E1 -19806.86,E2 -19806.86} C_VEL
LIN {X 0,Y 235.312,Z 621.167,A -85,B 0,C 180,E1 -19809.449,E2 -19809.449} C_VEL
LIN {X 0,Y 234.588,Z 621.263,A -85,B 0,C 180,E1 -19810.876,E2 -19810.876} C_VEL
LIN {X 0,Y 231.637,Z 621.624,A -85,B 0,C 180,E1 -19813.201,E2 -19813.201} C_VEL
LIN {X 0,Y 229.157,Z 621.936,A -85,B 0,C 180,E1 -19815.098,E2 -19815.098} C_VEL
LIN {X 0,Y 228.108,Z 622.064,A -85,B 0,C 180,E1 -19816.572,E2 -19816.572} C_VEL
LIN {X 0,Y 228.03,Z 622.077,A -85,B 0,C 180,E1 -19817.072,E2 -19817.072} C_VEL
LIN {X 0,Y 227.959,Z 622.084,A -85,B 0,C 180,E1 -19821.714,E2 -19821.714} C_VEL
LIN {X 0,Y 227.939,Z 622.084,A -85,B 0,C 180,E1 -19826.604,E2 -19826.604} C_VEL
LIN {X 0,Y 227.895,Z 622.093,A -85,B 0,C 180,E1 -19830.292,E2 -19830.292} C_VEL
LIN {X 0,Y 227.919,Z 622.159,A -85,B 0,C 180,E1 -19835.323,E2 -19835.323} C_VEL
LIN {X 0,Y 229.132,Z 626.081,A -85,B 0,C 180,E1 -19839.341,E2 -19839.341} C_VEL
LIN {X 0,Y 230.541,Z 630.328,A -85,B 0,C 180,E1 -19842.978,E2 -19842.978} C_VEL
LIN {X 0,Y 231.437,Z 633.257,A -85,B 0,C 180,E1 -19844.996,E2 -19844.996} C_VEL
LIN {X 0,Y 234.475,Z 638.104,A -85,B 0,C 180,E1 -19846.497,E2 -19846.497} C_VEL
LIN {X 0,Y 235.997,Z 640.236,A -85,B 0,C 180,E1 -19847.183,E2 -19847.183} C_VEL
LIN {X 0,Y 239.846,Z 646.466,A -85,B 0,C 180,E1 -19848.851,E2 -19848.851} C_VEL
LIN {X 0,Y 243.116,Z 652.202,A -85,B 0,C 180,E1 -19850.179,E2 -19850.179} C_VEL
LIN {X 0,Y 247.603,Z 660.696,A -85,B 0,C 180,E1 -19851.881,E2 -19851.881} C_VEL
LIN {X 0,Y 253.067,Z 672.736,A -85,B 0,C 180,E1 -19853.841,E2 -19853.841} C_VEL
LIN {X 0,Y 254.508,Z 676.721,A -85,B 0,C 180,E1 -19854.364,E2 -19854.364} C_VEL
LIN {X 0,Y 256.237,Z 692.666,A -85,B 0,C 180,E1 -19855.5,E2 -19855.5} C_VEL
LIN {X 0,Y 256.3,Z 698.424,A -85,B 0,C 180,E1 -19855.775,E2 -19855.775} C_VEL
LIN {X 0,Y 253.22,Z 744.963,A -85,B 0,C 180,E1 -19857.309,E2 -19857.309} C_VEL
LIN {X 0,Y 251.478,Z 758.896,A -85,B 0,C 180,E1 -19858.047,E2 -19858.047} C_VEL
LIN {X 0,Y 249.122,Z 771.638,A -85,B 0,C 180,E1 -19859.013,E2 -19859.013} C_VEL
LIN {X 0,Y 246.428,Z 783.783,A -85,B 0,C 180,E1 -19860.296,E2 -19860.296} C_VEL
LIN {X 0,Y 243.511,Z 794.81,A -85,B 0,C 180,E1 -19861.798,E2 -19861.798} C_VEL
LIN {X 0,Y 240.51,Z 804.871,A -85,B 0,C 180,E1 -19863.537,E2 -19863.537} C_VEL
LIN {X 0,Y 237.492,Z 814.061,A -85,B 0,C 180,E1 -19865.526,E2 -19865.526} C_VEL
LIN {X 0,Y 234.395,Z 823.089,A -85,B 0,C 180,E1 -19867.989,E2 -19867.989} C_VEL
LIN {X 0,Y 231.836,Z 830.411,A -85,B 0,C 180,E1 -19870.522,E2 -19870.522} C_VEL
LIN {X 0,Y 229.728,Z 836.312,A -85,B 0,C 180,E1 -19873.105,E2 -19873.105} C_VEL
LIN {X 0,Y 227.918,Z 841.01,A -85,B 0,C 180,E1 -19875.719,E2 -19875.719} C_VEL
LIN {X 0,Y 226.815,Z 844.64,A -85,B 0,C 180,E1 -19878.381,E2 -19878.381} C_VEL
LIN {X 0,Y 226.091,Z 847.277,A -85,B 0,C 180,E1 -19881.059,E2 -19881.059} C_VEL
LIN {X 0,Y 225.832,Z 848.51,A -85,B 0,C 180,E1 -19882.849,E2 -19882.849} C_VEL
LIN {X 0,Y 225.727,Z 849.473,A -85,B 0,C 180,E1 -19885.091,E2 -19885.091} C_VEL
LIN {X 0,Y 225.842,Z 849.779,A -85,B 0,C 180,E1 -19888.217,E2 -19888.217} C_VEL
LIN {X 0,Y 225.896,Z 849.376,A -85,B 0,C 180,E1 -19890,E2 -19890} C_VEL
LIN {X 0,Y 225.867,Z 848.523,A -85,B 0,C 180,E1 -19891.783,E2 -19891.783} C_VEL
LIN {X 0,Y 225.808,Z 847.25,A -85,B 0,C 180,E1 -19893.569,E2 -19893.569} C_VEL
LIN {X 0,Y 225.832,Z 844.483,A -85,B 0,C 180,E1 -19896.253,E2 -19896.253} C_VEL
LIN {X 0,Y 226.13,Z 840.632,A -85,B 0,C 180,E1 -19898.94,E2 -19898.94} C_VEL
LIN {X 0,Y 226.716,Z 835.585,A -85,B 0,C 180,E1 -19901.624,E2 -19901.624} C_VEL
LIN {X 0,Y 227.763,Z 829.208,A -85,B 0,C 180,E1 -19904.291,E2 -19904.291} C_VEL
LIN {X 0,Y 229.213,Z 821.171,A -85,B 0,C 180,E1 -19906.934,E2 -19906.934} C_VEL
LIN {X 0,Y 230.352,Z 814.135,A -85,B 0,C 180,E1 -19908.838,E2 -19908.838} C_VEL
LIN {X 0,Y 232.295,Z 803.996,A -85,B 0,C 180,E1 -19911.055,E2 -19911.055} C_VEL
LIN {X 0,Y 234.274,Z 793.083,A -85,B 0,C 180,E1 -19912.953,E2 -19912.953} C_VEL
LIN {X 0,Y 236.013,Z 782.46,A -85,B 0,C 180,E1 -19914.404,E2 -19914.404} C_VEL
LIN {X 0,Y 237.781,Z 769.814,A -85,B 0,C 180,E1 -19915.728,E2 -19915.728} C_VEL
LIN {X 0,Y 239.277,Z 756.571,A -85,B 0,C 180,E1 -19916.727,E2 -19916.727} C_VEL
LIN {X 0,Y 240.143,Z 743.256,A -85,B 0,C 180,E1 -19917.388,E2 -19917.388} C_VEL
LIN {X 0,Y 242.2,Z 692.177,A -85,B 0,C 180,E1 -19919.088,E2 -19919.088} C_VEL
LIN {X 0,Y 237.616,Z 655.538,A -85,B 0,C 180,E1 -19920.935,E2 -19920.935} C_VEL
LIN {X 0,Y 231.29,Z 637.905,A -85,B 0,C 180,E1 -19922.341,E2 -19922.341} C_VEL
LIN {X 0,Y 229.3,Z 628.158,A -85,B 0,C 180,E1 -19926.288,E2 -19926.288} C_VEL
LIN {X 0,Y 227.934,Z 622.094,A -85,B 0,C 180,E1 -19928.876,E2 -19928.876} C_VEL
LIN {X 0,Y 227.9,Z 622.101,A -85,B 0,C 180,E1 -19932.72,E2 -19932.72} C_VEL
LIN {X 0,Y 227.893,Z 622.097,A -85,B 0,C 180,E1 -19937.741,E2 -19937.741} C_VEL
LIN {X 0,Y 227.87,Z 622.099,A -85,B 0,C 180,E1 -19941.913,E2 -19941.913} C_VEL
LIN {X 0,Y 227.889,Z 622.098,A -85,B 0,C 180,E1 -19946.372,E2 -19946.372} C_VEL
LIN {X 0,Y 227.917,Z 622.093,A -85,B 0,C 180,E1 -19950.437,E2 -19950.437} C_VEL
LIN {X 0,Y 227.922,Z 622.089,A -85,B 0,C 180,E1 -19954.424,E2 -19954.424} C_VEL
LIN {X 0,Y 227.944,Z 622.091,A -85,B 0,C 180,E1 -19958.284,E2 -19958.284} C_VEL
LIN {X 0,Y 228.031,Z 622.076,A -85,B 0,C 180,E1 -19962.825,E2 -19962.825} C_VEL
LIN {X 0,Y 228.069,Z 622.074,A -85,B 0,C 180,E1 -19967.542,E2 -19967.542} C_VEL
LIN {X 0,Y 228.3,Z 622.039,A -85,B 0,C 180,E1 -19971.145,E2 -19971.145} C_VEL
LIN {X 0,Y 228.349,Z 622.037,A -85,B 0,C 180,E1 -19972.927,E2 -19972.927} C_VEL
LIN {X 0,Y 228.55,Z 622.011,A -85,B 0,C 180,E1 -19978.237,E2 -19978.237} C_VEL
LIN {X 0,Y 228.55,Z 622.007,A -85,B 0,C 180,E1 -19981.761,E2 -19981.761} C_VEL
LIN {X 0,Y 228.348,Z 622.04,A -85,B 0,C 180,E1 -19987.071,E2 -19987.071} C_VEL
LIN {X 0,Y 228.153,Z 622.058,A -85,B 0,C 180,E1 -19990.65,E2 -19990.65} C_VEL
LIN {X 0,Y 228.054,Z 622.068,A -85,B 0,C 180,E1 -19994.272,E2 -19994.272} C_VEL
LIN {X 0,Y 227.997,Z 622.084,A -85,B 0,C 180,E1 -19997.953,E2 -19997.953} C_VEL
LIN {X 0,Y 227.924,Z 622.087,A -85,B 0,C 180,E1 -20002.328,E2 -20002.328} C_VEL
LIN {X 0,Y 227.936,Z 622.081,A -85,B 0,C 180,E1 -20006.602,E2 -20006.602} C_VEL
LIN {X 0,Y 227.891,Z 622.097,A -85,B 0,C 180,E1 -20010.291,E2 -20010.291} C_VEL
LIN {X 0,Y 227.885,Z 622.097,A -85,B 0,C 180,E1 -20013.718,E2 -20013.718} C_VEL
LIN {X 0,Y 227.866,Z 622.089,A -85,B 0,C 180,E1 -20018.086,E2 -20018.086} C_VEL
LIN {X 0,Y 227.904,Z 622.095,A -85,B 0,C 180,E1 -20022.719,E2 -20022.719} C_VEL
LIN {X 0,Y 227.892,Z 622.092,A -85,B 0,C 180,E1 -20027.742,E2 -20027.742} C_VEL
LIN {X 0,Y 227.866,Z 622.096,A -85,B 0,C 180,E1 -20031.914,E2 -20031.914} C_VEL
LIN {X 0,Y 227.886,Z 622.099,A -85,B 0,C 180,E1 -20036.373,E2 -20036.373} C_VEL
LIN {X 0,Y 227.9,Z 622.09,A -85,B 0,C 180,E1 -20040.436,E2 -20040.436} C_VEL
LIN {X 0,Y 227.924,Z 622.095,A -85,B 0,C 180,E1 -20044.426,E2 -20044.426} C_VEL
LIN {X 0,Y 227.959,Z 622.089,A -85,B 0,C 180,E1 -20048.287,E2 -20048.287} C_VEL
LIN {X 0,Y 228.031,Z 622.08,A -85,B 0,C 180,E1 -20052.826,E2 -20052.826} C_VEL
LIN {X 0,Y 228.091,Z 622.07,A -85,B 0,C 180,E1 -20057.545,E2 -20057.545} C_VEL
LIN {X 0,Y 228.302,Z 622.044,A -85,B 0,C 180,E1 -20061.146,E2 -20061.146} C_VEL
LIN {X 0,Y 228.351,Z 622.039,A -85,B 0,C 180,E1 -20062.929,E2 -20062.929} C_VEL
LIN {X 0,Y 228.552,Z 622.012,A -85,B 0,C 180,E1 -20068.238,E2 -20068.238} C_VEL
LIN {X 0,Y 228.552,Z 622.013,A -85,B 0,C 180,E1 -20071.762,E2 -20071.762} C_VEL
LIN {X 0,Y 228.336,Z 622.044,A -85,B 0,C 180,E1 -20077.072,E2 -20077.072} C_VEL
LIN {X 0,Y 228.143,Z 622.067,A -85,B 0,C 180,E1 -20080.651,E2 -20080.651} C_VEL
LIN {X 0,Y 228.096,Z 622.276,A -85,B 0,C 180,E1 -20082.608,E2 -20082.608} C_VEL
LIN {X 0,Y 230.042,Z 627.033,A -85,B 0,C 180,E1 -20083.029,E2 -20083.029} C_VEL
LIN {X 0,Y 238.462,Z 645.693,A -85,B 0,C 180,E1 -20084.698,E2 -20084.698} C_VEL
LIN {X 0,Y 243.186,Z 659.183,A -85,B 0,C 180,E1 -20085.688,E2 -20085.688} C_VEL
LIN {X 0,Y 240.281,Z 725.016,A -85,B 0,C 180,E1 -20087.885,E2 -20087.885} C_VEL
LIN {X 0,Y 239.305,Z 738.957,A -85,B 0,C 180,E1 -20088.708,E2 -20088.708} C_VEL
LIN {X 0,Y 237.999,Z 751.605,A -85,B 0,C 180,E1 -20089.798,E2 -20089.798} C_VEL
LIN {X 0,Y 236.292,Z 764.766,A -85,B 0,C 180,E1 -20091.342,E2 -20091.342} C_VEL
LIN {X 0,Y 234.618,Z 775.224,A -85,B 0,C 180,E1 -20092.918,E2 -20092.918} C_VEL
LIN {X 0,Y 232.701,Z 786.292,A -85,B 0,C 180,E1 -20095.037,E2 -20095.037} C_VEL
LIN {X 0,Y 231.085,Z 795.126,A -85,B 0,C 180,E1 -20097.141,E2 -20097.141} C_VEL
LIN {X 0,Y 229.429,Z 803.695,A -85,B 0,C 180,E1 -20099.666,E2 -20099.666} C_VEL
LIN {X 0,Y 228.012,Z 811.294,A -85,B 0,C 180,E1 -20102.524,E2 -20102.524} C_VEL
LIN {X 0,Y 226.979,Z 817.436,A -85,B 0,C 180,E1 -20105.489,E2 -20105.489} C_VEL
LIN {X 0,Y 226.159,Z 822.007,A -85,B 0,C 180,E1 -20108.425,E2 -20108.425} C_VEL
LIN {X 0,Y 225.628,Z 825.491,A -85,B 0,C 180,E1 -20111.621,E2 -20111.621} C_VEL
LIN {X 0,Y 225.46,Z 827.304,A -85,B 0,C 180,E1 -20114.198,E2 -20114.198} C_VEL
LIN {X 0,Y 225.526,Z 828.262,A -85,B 0,C 180,E1 -20116.72,E2 -20116.72} C_VEL
LIN {X 0,Y 225.87,Z 828.389,A -85,B 0,C 180,E1 -20119.201,E2 -20119.201} C_VEL
LIN {X 0,Y 226.456,Z 827.75,A -85,B 0,C 180,E1 -20121.634,E2 -20121.634} C_VEL
LIN {X 0,Y 227.234,Z 826.413,A -85,B 0,C 180,E1 -20124.011,E2 -20124.011} C_VEL
LIN {X 0,Y 228.862,Z 823.058,A -85,B 0,C 180,E1 -20127.494,E2 -20127.494} C_VEL
LIN {X 0,Y 230.382,Z 819.651,A -85,B 0,C 180,E1 -20129.914,E2 -20129.914} C_VEL
LIN {X 0,Y 232.256,Z 815.176,A -85,B 0,C 180,E1 -20132.365,E2 -20132.365} C_VEL
LIN {X 0,Y 234.966,Z 808.368,A -85,B 0,C 180,E1 -20135.245,E2 -20135.245} C_VEL
LIN {X 0,Y 238.075,Z 800.104,A -85,B 0,C 180,E1 -20137.891,E2 -20137.891} C_VEL
LIN {X 0,Y 241.162,Z 790.948,A -85,B 0,C 180,E1 -20140.208,E2 -20140.208} C_VEL
LIN {X 0,Y 244.158,Z 781.016,A -85,B 0,C 180,E1 -20142.188,E2 -20142.188} C_VEL
LIN {X 0,Y 247.079,Z 769.915,A -85,B 0,C 180,E1 -20143.922,E2 -20143.922} C_VEL
LIN {X 0,Y 249.699,Z 758.3,A -85,B 0,C 180,E1 -20145.327,E2 -20145.327} C_VEL
LIN {X 0,Y 251.838,Z 745.81,A -85,B 0,C 180,E1 -20146.472,E2 -20146.472} C_VEL
LIN {X 0,Y 253.318,Z 733.656,A -85,B 0,C 180,E1 -20147.294,E2 -20147.294} C_VEL
LIN {X 0,Y 254.496,Z 720.657,A -85,B 0,C 180,E1 -20147.846,E2 -20147.846} C_VEL
LIN {X 0,Y 257.707,Z 670.776,A -85,B 0,C 180,E1 -20149.47,E2 -20149.47} C_VEL
LIN {X 0,Y 252.632,Z 659.706,A -85,B 0,C 180,E1 -20151.169,E2 -20151.169} C_VEL
LIN {X 0,Y 246.603,Z 648.801,A -85,B 0,C 180,E1 -20153.295,E2 -20153.295} C_VEL
LIN {X 0,Y 242.313,Z 641.845,A -85,B 0,C 180,E1 -20154.921,E2 -20154.921} C_VEL
LIN {X 0,Y 238.994,Z 637.12,A -85,B 0,C 180,E1 -20156.26,E2 -20156.26} C_VEL
LIN {X 0,Y 236.266,Z 633.201,A -85,B 0,C 180,E1 -20157.444,E2 -20157.444} C_VEL
LIN {X 0,Y 233.257,Z 629.142,A -85,B 0,C 180,E1 -20158.838,E2 -20158.838} C_VEL
LIN {X 0,Y 232.138,Z 627.542,A -85,B 0,C 180,E1 -20159.396,E2 -20159.396} C_VEL
LIN {X 0,Y 229.493,Z 624.691,A -85,B 0,C 180,E1 -20160.714,E2 -20160.714} C_VEL
LIN {X 0,Y 228.774,Z 623.079,A -85,B 0,C 180,E1 -20161.211,E2 -20161.211} C_VEL
LIN {X 0,Y 228.365,Z 622.04,A -85,B 0,C 180,E1 -20162.647,E2 -20162.647} C_VEL
LIN {X 0,Y 228.351,Z 622.035,A -85,B 0,C 180,E1 -20167.072,E2 -20167.072} C_VEL
LIN {X 0,Y 228.155,Z 622.061,A -85,B 0,C 180,E1 -20170.652,E2 -20170.652} C_VEL
LIN {X 0,Y 228.059,Z 622.078,A -85,B 0,C 180,E1 -20174.273,E2 -20174.273} C_VEL
LIN {X 0,Y 228.03,Z 622.077,A -85,B 0,C 180,E1 -20177.072,E2 -20177.072} C_VEL
LIN {X 0,Y 227.369,Z 622.17,A -85,B 0,C 180,E1 -20178.545,E2 -20178.545} C_VEL
LIN {X 0,Y 224.481,Z 622.535,A -85,B 0,C 180,E1 -20180.947,E2 -20180.947} C_VEL
LIN {X 0,Y 222.009,Z 622.836,A -85,B 0,C 180,E1 -20182.907,E2 -20182.907} C_VEL
LIN {X 0,Y 220.938,Z 622.961,A -85,B 0,C 180,E1 -20184.43,E2 -20184.43} C_VEL
LIN {X 0,Y 220.846,Z 622.968,A -85,B 0,C 180,E1 -20184.947,E2 -20184.947} C_VEL
LIN {X 0,Y 220.825,Z 622.967,A -85,B 0,C 180,E1 -20188.516,E2 -20188.516} C_VEL
LIN {X 0,Y 220.845,Z 623.135,A -85,B 0,C 180,E1 -20191.406,E2 -20191.406} C_VEL
LIN {X 0,Y 221.723,Z 625.51,A -85,B 0,C 180,E1 -20194.79,E2 -20194.79} C_VEL
LIN {X 0,Y 222.962,Z 629.463,A -85,B 0,C 180,E1 -20199.082,E2 -20199.082} C_VEL
LIN {X 0,Y 223.901,Z 632.331,A -85,B 0,C 180,E1 -20201.537,E2 -20201.537} C_VEL
LIN {X 0,Y 227.502,Z 637.84,A -85,B 0,C 180,E1 -20203.695,E2 -20203.695} C_VEL
LIN {X 0,Y 228.74,Z 639.465,A -85,B 0,C 180,E1 -20204.347,E2 -20204.347} C_VEL
LIN {X 0,Y 233.005,Z 646.106,A -85,B 0,C 180,E1 -20206.502,E2 -20206.502} C_VEL
LIN {X 0,Y 236.524,Z 651.976,A -85,B 0,C 180,E1 -20208.112,E2 -20208.112} C_VEL
LIN {X 0,Y 239.772,Z 657.921,A -85,B 0,C 180,E1 -20209.514,E2 -20209.514} C_VEL
LIN {X 0,Y 243.534,Z 665.223,A -85,B 0,C 180,E1 -20211.022,E2 -20211.022} C_VEL
LIN {X 0,Y 248.56,Z 676.654,A -85,B 0,C 180,E1 -20212.96,E2 -20212.96} C_VEL
LIN {X 0,Y 249.654,Z 679.718,A -85,B 0,C 180,E1 -20213.378,E2 -20213.378} C_VEL
LIN {X 0,Y 251.178,Z 694.788,A -85,B 0,C 180,E1 -20214.475,E2 -20214.475} C_VEL
LIN {X 0,Y 251.07,Z 700.313,A -85,B 0,C 180,E1 -20214.719,E2 -20214.719} C_VEL
LIN {X 0,Y 247.945,Z 744.559,A -85,B 0,C 180,E1 -20216.213,E2 -20216.213} C_VEL
LIN {X 0,Y 246.133,Z 758.461,A -85,B 0,C 180,E1 -20216.964,E2 -20216.964} C_VEL
LIN {X 0,Y 243.771,Z 770.721,A -85,B 0,C 180,E1 -20217.89,E2 -20217.89} C_VEL
LIN {X 0,Y 240.762,Z 783.745,A -85,B 0,C 180,E1 -20219.281,E2 -20219.281} C_VEL
LIN {X 0,Y 237.701,Z 794.721,A -85,B 0,C 180,E1 -20220.802,E2 -20220.802} C_VEL
LIN {X 0,Y 234.22,Z 805.693,A -85,B 0,C 180,E1 -20222.769,E2 -20222.769} C_VEL
LIN {X 0,Y 231.092,Z 814.657,A -85,B 0,C 180,E1 -20224.801,E2 -20224.801} C_VEL
LIN {X 0,Y 227.836,Z 823.486,A -85,B 0,C 180,E1 -20227.321,E2 -20227.321} C_VEL
LIN {X 0,Y 225.164,Z 830.625,A -85,B 0,C 180,E1 -20229.92,E2 -20229.92} C_VEL
LIN {X 0,Y 222.938,Z 836.404,A -85,B 0,C 180,E1 -20232.574,E2 -20232.574} C_VEL
LIN {X 0,Y 221.03,Z 841.001,A -85,B 0,C 180,E1 -20235.264,E2 -20235.264} C_VEL
LIN {X 0,Y 219.823,Z 844.534,A -85,B 0,C 180,E1 -20238.006,E2 -20238.006} C_VEL
LIN {X 0,Y 219.047,Z 847.092,A -85,B 0,C 180,E1 -20240.769,E2 -20240.769} C_VEL
LIN {X 0,Y 218.648,Z 849.032,A -85,B 0,C 180,E1 -20244.467,E2 -20244.467} C_VEL
LIN {X 0,Y 218.633,Z 849.416,A -85,B 0,C 180,E1 -20246.314,E2 -20246.314} C_VEL
LIN {X 0,Y 218.771,Z 849.397,A -85,B 0,C 180,E1 -20248.159,E2 -20248.159} C_VEL
LIN {X 0,Y 218.826,Z 848.922,A -85,B 0,C 180,E1 -20250,E2 -20250} C_VEL
LIN {X 0,Y 218.798,Z 848.028,A -85,B 0,C 180,E1 -20251.841,E2 -20251.841} C_VEL
LIN {X 0,Y 218.726,Z 845.416,A -85,B 0,C 180,E1 -20255.067,E2 -20255.067} C_VEL
LIN {X 0,Y 218.959,Z 841.357,A -85,B 0,C 180,E1 -20258.305,E2 -20258.305} C_VEL
LIN {X 0,Y 219.483,Z 836.608,A -85,B 0,C 180,E1 -20261.076,E2 -20261.076} C_VEL
LIN {X 0,Y 220.606,Z 829.409,A -85,B 0,C 180,E1 -20264.294,E2 -20264.294} C_VEL
LIN {X 0,Y 222.066,Z 821.551,A -85,B 0,C 180,E1 -20267.022,E2 -20267.022} C_VEL
LIN {X 0,Y 223.004,Z 815.849,A -85,B 0,C 180,E1 -20268.658,E2 -20268.658} C_VEL
LIN {X 0,Y 225.084,Z 805.793,A -85,B 0,C 180,E1 -20271.043,E2 -20271.043} C_VEL
LIN {X 0,Y 226.789,Z 796.612,A -85,B 0,C 180,E1 -20272.79,E2 -20272.79} C_VEL
LIN {X 0,Y 228.756,Z 785.327,A -85,B 0,C 180,E1 -20274.503,E2 -20274.503} C_VEL
LIN {X 0,Y 230.37,Z 774.716,A -85,B 0,C 180,E1 -20275.767,E2 -20275.767} C_VEL
LIN {X 0,Y 231.971,Z 762.096,A -85,B 0,C 180,E1 -20276.907,E2 -20276.907} C_VEL
LIN {X 0,Y 233.178,Z 748.807,A -85,B 0,C 180,E1 -20277.728,E2 -20277.728} C_VEL
LIN {X 0,Y 234.327,Z 724.778,A -85,B 0,C 180,E1 -20278.615,E2 -20278.615} C_VEL
LIN {X 0,Y 235.519,Z 692.092,A -85,B 0,C 180,E1 -20279.747,E2 -20279.747} C_VEL
LIN {X 0,Y 231.226,Z 657.511,A -85,B 0,C 180,E1 -20281.54,E2 -20281.54} C_VEL
LIN {X 0,Y 224.008,Z 637.496,A -85,B 0,C 180,E1 -20283.233,E2 -20283.233} C_VEL
LIN {X 0,Y 222.198,Z 628.707,A -85,B 0,C 180,E1 -20286.938,E2 -20286.938} C_VEL
LIN {X 0,Y 220.857,Z 622.977,A -85,B 0,C 180,E1 -20289.525,E2 -20289.525} C_VEL
LIN {X 0,Y 220.86,Z 622.977,A -85,B 0,C 180,E1 -20292.954,E2 -20292.954} C_VEL
LIN {X 0,Y 220.839,Z 622.976,A -85,B 0,C 180,E1 -20298.062,E2 -20298.062} C_VEL
LIN {X 0,Y 220.837,Z 622.979,A -85,B 0,C 180,E1 -20302.711,E2 -20302.711} C_VEL
LIN {X 0,Y 220.823,Z 622.979,A -85,B 0,C 180,E1 -20307.244,E2 -20307.244} C_VEL
LIN {X 0,Y 220.834,Z 622.976,A -85,B 0,C 180,E1 -20311.485,E2 -20311.485} C_VEL
LIN {X 0,Y 220.859,Z 622.972,A -85,B 0,C 180,E1 -20315.563,E2 -20315.563} C_VEL
LIN {X 0,Y 220.881,Z 622.969,A -85,B 0,C 180,E1 -20319.512,E2 -20319.512} C_VEL
LIN {X 0,Y 221.012,Z 622.954,A -85,B 0,C 180,E1 -20323.369,E2 -20323.369} C_VEL
LIN {X 0,Y 221.102,Z 622.94,A -85,B 0,C 180,E1 -20329.004,E2 -20329.004} C_VEL
LIN {X 0,Y 221.284,Z 622.916,A -85,B 0,C 180,E1 -20332.7,E2 -20332.7} C_VEL
LIN {X 0,Y 221.508,Z 622.888,A -85,B 0,C 180,E1 -20338.181,E2 -20338.181} C_VEL
LIN {X 0,Y 221.508,Z 622.884,A -85,B 0,C 180,E1 -20341.817,E2 -20341.817} C_VEL
LIN {X 0,Y 221.299,Z 622.919,A -85,B 0,C 180,E1 -20347.297,E2 -20347.297} C_VEL
LIN {X 0,Y 221.101,Z 622.936,A -85,B 0,C 180,E1 -20350.994,E2 -20350.994} C_VEL
LIN {X 0,Y 221.009,Z 622.949,A -85,B 0,C 180,E1 -20356.629,E2 -20356.629} C_VEL
LIN {X 0,Y 220.886,Z 622.967,A -85,B 0,C 180,E1 -20360.486,E2 -20360.486} C_VEL
LIN {X 0,Y 220.861,Z 622.959,A -85,B 0,C 180,E1 -20364.435,E2 -20364.435} C_VEL
LIN {X 0,Y 220.822,Z 622.973,A -85,B 0,C 180,E1 -20368.515,E2 -20368.515} C_VEL
LIN {X 0,Y 220.818,Z 622.976,A -85,B 0,C 180,E1 -20372.755,E2 -20372.755} C_VEL
LIN {X 0,Y 220.833,Z 622.964,A -85,B 0,C 180,E1 -20377.288,E2 -20377.288} C_VEL
LIN {X 0,Y 220.848,Z 622.972,A -85,B 0,C 180,E1 -20381.933,E2 -20381.933} C_VEL
LIN {X 0,Y 220.857,Z 622.968,A -85,B 0,C 180,E1 -20387.044,E2 -20387.044} C_VEL
LIN {X 0,Y 220.808,Z 622.971,A -85,B 0,C 180,E1 -20390.465,E2 -20390.465} C_VEL
LIN {X 0,Y 220.83,Z 622.977,A -85,B 0,C 180,E1 -20392.795,E2 -20392.795} C_VEL
LIN {X 0,Y 220.819,Z 622.974,A -85,B 0,C 180,E1 -20397.245,E2 -20397.245} C_VEL
LIN {X 0,Y 220.823,Z 622.974,A -85,B 0,C 180,E1 -20401.485,E2 -20401.485} C_VEL
LIN {X 0,Y 220.864,Z 622.97,A -85,B 0,C 180,E1 -20405.565,E2 -20405.565} C_VEL
LIN {X 0,Y 220.889,Z 622.967,A -85,B 0,C 180,E1 -20409.514,E2 -20409.514} C_VEL
LIN {X 0,Y 221.013,Z 622.952,A -85,B 0,C 180,E1 -20413.37,E2 -20413.37} C_VEL
LIN {X 0,Y 221.109,Z 622.94,A -85,B 0,C 180,E1 -20419.006,E2 -20419.006} C_VEL
LIN {X 0,Y 221.286,Z 622.918,A -85,B 0,C 180,E1 -20422.702,E2 -20422.702} C_VEL
LIN {X 0,Y 221.51,Z 622.889,A -85,B 0,C 180,E1 -20428.182,E2 -20428.182} C_VEL
LIN {X 0,Y 221.51,Z 622.89,A -85,B 0,C 180,E1 -20431.818,E2 -20431.818} C_VEL
LIN {X 0,Y 221.268,Z 622.924,A -85,B 0,C 180,E1 -20437.299,E2 -20437.299} C_VEL
LIN {X 0,Y 221.049,Z 622.95,A -85,B 0,C 180,E1 -20441.751,E2 -20441.751} C_VEL
LIN {X 0,Y 222.171,Z 626.014,A -85,B 0,C 180,E1 -20442.036,E2 -20442.036} C_VEL
LIN {X 0,Y 230.708,Z 644.818,A -85,B 0,C 180,E1 -20443.82,E2 -20443.82} C_VEL
LIN {X 0,Y 234.082,Z 653.453,A -85,B 0,C 180,E1 -20444.53,E2 -20444.53} C_VEL
LIN {X 0,Y 236.605,Z 660.89,A -85,B 0,C 180,E1 -20445.083,E2 -20445.083} C_VEL
LIN {X 0,Y 233.623,Z 725.336,A -85,B 0,C 180,E1 -20447.299,E2 -20447.299} C_VEL
LIN {X 0,Y 232.586,Z 739.458,A -85,B 0,C 180,E1 -20448.156,E2 -20448.156} C_VEL
LIN {X 0,Y 231.171,Z 752.497,A -85,B 0,C 180,E1 -20449.321,E2 -20449.321} C_VEL
LIN {X 0,Y 229.496,Z 765.133,A -85,B 0,C 180,E1 -20450.854,E2 -20450.854} C_VEL
LIN {X 0,Y 227.672,Z 776.109,A -85,B 0,C 180,E1 -20452.565,E2 -20452.565} C_VEL
LIN {X 0,Y 225.855,Z 786.224,A -85,B 0,C 180,E1 -20454.556,E2 -20454.556} C_VEL
LIN {X 0,Y 224.143,Z 795.379,A -85,B 0,C 180,E1 -20456.79,E2 -20456.79} C_VEL
LIN {X 0,Y 222.462,Z 803.764,A -85,B 0,C 180,E1 -20459.318,E2 -20459.318} C_VEL
LIN {X 0,Y 221.209,Z 810.448,A -85,B 0,C 180,E1 -20461.839,E2 -20461.839} C_VEL
LIN {X 0,Y 219.97,Z 817.216,A -85,B 0,C 180,E1 -20465.105,E2 -20465.105} C_VEL
LIN {X 0,Y 219.298,Z 821.069,A -85,B 0,C 180,E1 -20467.509,E2 -20467.509} C_VEL
LIN {X 0,Y 218.764,Z 824.16,A -85,B 0,C 180,E1 -20469.979,E2 -20469.979} C_VEL
LIN {X 0,Y 218.446,Z 826.479,A -85,B 0,C 180,E1 -20472.501,E2 -20472.501} C_VEL
LIN {X 0,Y 218.364,Z 827.988,A -85,B 0,C 180,E1 -20475.076,E2 -20475.076} C_VEL
LIN {X 0,Y 218.52,Z 828.717,A -85,B 0,C 180,E1 -20477.706,E2 -20477.706} C_VEL
LIN {X 0,Y 219.026,Z 828.63,A -85,B 0,C 180,E1 -20480.361,E2 -20480.361} C_VEL
LIN {X 0,Y 219.805,Z 827.686,A -85,B 0,C 180,E1 -20483.066,E2 -20483.066} C_VEL
LIN {X 0,Y 220.898,Z 825.814,A -85,B 0,C 180,E1 -20485.811,E2 -20485.811} C_VEL
LIN {X 0,Y 222.374,Z 822.922,A -85,B 0,C 180,E1 -20488.572,E2 -20488.572} C_VEL
LIN {X 0,Y 224.764,Z 817.678,A -85,B 0,C 180,E1 -20492.03,E2 -20492.03} C_VEL
LIN {X 0,Y 227.373,Z 811.845,A -85,B 0,C 180,E1 -20494.85,E2 -20494.85} C_VEL
LIN {X 0,Y 230.593,Z 804.038,A -85,B 0,C 180,E1 -20497.724,E2 -20497.724} C_VEL
LIN {X 0,Y 233.678,Z 795.808,A -85,B 0,C 180,E1 -20500.091,E2 -20500.091} C_VEL
LIN {X 0,Y 236.833,Z 786.638,A -85,B 0,C 180,E1 -20502.181,E2 -20502.181} C_VEL
LIN {X 0,Y 239.798,Z 776.59,A -85,B 0,C 180,E1 -20504.001,E2 -20504.001} C_VEL
LIN {X 0,Y 242.622,Z 765.796,A -85,B 0,C 180,E1 -20505.533,E2 -20505.533} C_VEL
LIN {X 0,Y 245.1,Z 754.173,A -85,B 0,C 180,E1 -20506.835,E2 -20506.835} C_VEL
LIN {X 0,Y 247.189,Z 740.873,A -85,B 0,C 180,E1 -20507.949,E2 -20507.949} C_VEL
LIN {X 0,Y 248.595,Z 728.507,A -85,B 0,C 180,E1 -20508.662,E2 -20508.662} C_VEL
LIN {X 0,Y 252.51,Z 673.195,A -85,B 0,C 180,E1 -20510.532,E2 -20510.532} C_VEL
LIN {X 0,Y 248.153,Z 663.655,A -85,B 0,C 180,E1 -20512.084,E2 -20512.084} C_VEL
LIN {X 0,Y 242.096,Z 652.513,A -85,B 0,C 180,E1 -20514.36,E2 -20514.36} C_VEL
LIN {X 0,Y 238.844,Z 647.133,A -85,B 0,C 180,E1 -20515.692,E2 -20515.692} C_VEL
LIN {X 0,Y 235.613,Z 642.47,A -85,B 0,C 180,E1 -20517.062,E2 -20517.062} C_VEL
LIN {X 0,Y 232.274,Z 637.731,A -85,B 0,C 180,E1 -20518.614,E2 -20518.614} C_VEL
LIN {X 0,Y 229.337,Z 633.454,A -85,B 0,C 180,E1 -20520.111,E2 -20520.111} C_VEL
LIN {X 0,Y 226.835,Z 630.643,A -85,B 0,C 180,E1 -20521.443,E2 -20521.443} C_VEL
LIN {X 0,Y 225.879,Z 629.041,A -85,B 0,C 180,E1 -20522.029,E2 -20522.029} C_VEL
LIN {X 0,Y 222.396,Z 626.121,A -85,B 0,C 180,E1 -20524.078,E2 -20524.078} C_VEL
LIN {X 0,Y 221.383,Z 624.029,A -85,B 0,C 180,E1 -20524.895,E2 -20524.895} C_VEL
LIN {X 0,Y 221.252,Z 622.919,A -85,B 0,C 180,E1 -20526.613,E2 -20526.613} C_VEL
LIN {X 0,Y 221.185,Z 622.926,A -85,B 0,C 180,E1 -20529.943,E2 -20529.943} C_VEL
LIN {X 0,Y 220.991,Z 622.956,A -85,B 0,C 180,E1 -20534.74,E2 -20534.74} C_VEL
LIN {X 0,Y 220.919,Z 622.961,A -85,B 0,C 180,E1 -20538.551,E2 -20538.551} C_VEL
LIN {X 0,Y 220.893,Z 622.961,A -85,B 0,C 180,E1 -20542.684,E2 -20542.684} C_VEL
LIN {X 0,Y 220.846,Z 622.968,A -85,B 0,C 180,E1 -20544.947,E2 -20544.947} C_VEL
LIN {X 0,Y 220.234,Z 623.282,A -85,B 0,C 180,E1 -20546.468,E2 -20546.468} C_VEL
LIN {X 0,Y 217.741,Z 624.812,A -85,B 0,C 180,E1 -20548.943,E2 -20548.943} C_VEL
LIN {X 0,Y 215.761,Z 626.474,A -85,B 0,C 180,E1 -20550.949,E2 -20550.949} C_VEL
LIN {X 0,Y 215.096,Z 627.7,A -85,B 0,C 180,E1 -20552.495,E2 -20552.495} C_VEL
LIN {X 0,Y 215.137,Z 628.069,A -85,B 0,C 180,E1 -20553.016,E2 -20553.016} C_VEL
LIN {X 0,Y 216.213,Z 631.078,A -85,B 0,C 180,E1 -20556.822,E2 -20556.822} C_VEL
LIN {X 0,Y 220.438,Z 637.265,A -85,B 0,C 180,E1 -20560.151,E2 -20560.151} C_VEL
LIN {X 0,Y 221.745,Z 638.981,A -85,B 0,C 180,E1 -20561.026,E2 -20561.026} C_VEL
LIN {X 0,Y 225.592,Z 644.692,A -85,B 0,C 180,E1 -20563.388,E2 -20563.388} C_VEL
LIN {X 0,Y 229.92,Z 651.7,A -85,B 0,C 180,E1 -20565.72,E2 -20565.72} C_VEL
LIN {X 0,Y 233.244,Z 657.475,A -85,B 0,C 180,E1 -20567.351,E2 -20567.351} C_VEL
LIN {X 0,Y 237.863,Z 666.225,A -85,B 0,C 180,E1 -20569.419,E2 -20569.419} C_VEL
LIN {X 0,Y 242.563,Z 676.605,A -85,B 0,C 180,E1 -20571.38,E2 -20571.38} C_VEL
LIN {X 0,Y 244.901,Z 682.657,A -85,B 0,C 180,E1 -20572.338,E2 -20572.338} C_VEL
LIN {X 0,Y 246.202,Z 696.776,A -85,B 0,C 180,E1 -20573.403,E2 -20573.403} C_VEL
LIN {X 0,Y 244.419,Z 723.876,A -85,B 0,C 180,E1 -20574.345,E2 -20574.345} C_VEL
LIN {X 0,Y 242.686,Z 745.524,A -85,B 0,C 180,E1 -20575.115,E2 -20575.115} C_VEL
LIN {X 0,Y 240.88,Z 758.426,A -85,B 0,C 180,E1 -20575.831,E2 -20575.831} C_VEL
LIN {X 0,Y 238.545,Z 770.041,A -85,B 0,C 180,E1 -20576.721,E2 -20576.721} C_VEL
LIN {X 0,Y 235.583,Z 782.295,A -85,B 0,C 180,E1 -20578.028,E2 -20578.028} C_VEL
LIN {X 0,Y 232.369,Z 793.397,A -85,B 0,C 180,E1 -20579.563,E2 -20579.563} C_VEL
LIN {X 0,Y 228.603,Z 804.574,A -85,B 0,C 180,E1 -20581.542,E2 -20581.542} C_VEL
LIN {X 0,Y 225.342,Z 813.656,A -85,B 0,C 180,E1 -20583.614,E2 -20583.614} C_VEL
LIN {X 0,Y 221.836,Z 822.596,A -85,B 0,C 180,E1 -20586.176,E2 -20586.176} C_VEL
LIN {X 0,Y 219.25,Z 829.181,A -85,B 0,C 180,E1 -20588.576,E2 -20588.576} C_VEL
LIN {X 0,Y 216.866,Z 834.774,A -85,B 0,C 180,E1 -20591.091,E2 -20591.091} C_VEL
LIN {X 0,Y 214.796,Z 839.627,A -85,B 0,C 180,E1 -20593.853,E2 -20593.853} C_VEL
LIN {X 0,Y 213.198,Z 843.401,A -85,B 0,C 180,E1 -20596.659,E2 -20596.659} C_VEL
LIN {X 0,Y 212.515,Z 845.38,A -85,B 0,C 180,E1 -20598.556,E2 -20598.556} C_VEL
LIN {X 0,Y 212.023,Z 846.898,A -85,B 0,C 180,E1 -20600.46,E2 -20600.46} C_VEL
LIN {X 0,Y 211.57,Z 848.744,A -85,B 0,C 180,E1 -20604.281,E2 -20604.281} C_VEL
LIN {X 0,Y 211.547,Z 849.083,A -85,B 0,C 180,E1 -20606.19,E2 -20606.19} C_VEL
LIN {X 0,Y 211.699,Z 848.987,A -85,B 0,C 180,E1 -20608.098,E2 -20608.098} C_VEL
LIN {X 0,Y 211.758,Z 848.469,A -85,B 0,C 180,E1 -20610,E2 -20610} C_VEL
LIN {X 0,Y 211.729,Z 847.533,A -85,B 0,C 180,E1 -20611.902,E2 -20611.902} C_VEL
LIN {X 0,Y 211.638,Z 845.084,A -85,B 0,C 180,E1 -20614.967,E2 -20614.967} C_VEL
LIN {X 0,Y 211.798,Z 841.974,A -85,B 0,C 180,E1 -20617.627,E2 -20617.627} C_VEL
LIN {X 0,Y 212.253,Z 837.533,A -85,B 0,C 180,E1 -20620.493,E2 -20620.493} C_VEL
LIN {X 0,Y 213.05,Z 831.827,A -85,B 0,C 180,E1 -20623.35,E2 -20623.35} C_VEL
LIN {X 0,Y 214.446,Z 824.663,A -85,B 0,C 180,E1 -20626.174,E2 -20626.174} C_VEL
LIN {X 0,Y 215.84,Z 817.307,A -85,B 0,C 180,E1 -20628.51,E2 -20628.51} C_VEL
LIN {X 0,Y 216.862,Z 811.851,A -85,B 0,C 180,E1 -20629.975,E2 -20629.975} C_VEL
LIN {X 0,Y 218.745,Z 802.099,A -85,B 0,C 180,E1 -20632.179,E2 -20632.179} C_VEL
LIN {X 0,Y 220.631,Z 792.237,A -85,B 0,C 180,E1 -20633.962,E2 -20633.962} C_VEL
LIN {X 0,Y 222.523,Z 781.591,A -85,B 0,C 180,E1 -20635.487,E2 -20635.487} C_VEL
LIN {X 0,Y 224.4,Z 768.917,A -85,B 0,C 180,E1 -20636.882,E2 -20636.882} C_VEL
LIN {X 0,Y 225.894,Z 756.433,A -85,B 0,C 180,E1 -20637.881,E2 -20637.881} C_VEL
LIN {X 0,Y 226.843,Z 743.521,A -85,B 0,C 180,E1 -20638.572,E2 -20638.572} C_VEL
LIN {X 0,Y 228.957,Z 693.011,A -85,B 0,C 180,E1 -20640.371,E2 -20640.371} C_VEL
LIN {X 0,Y 224.909,Z 659.685,A -85,B 0,C 180,E1 -20642.162,E2 -20642.162} C_VEL
LIN {X 0,Y 217.376,Z 639.314,A -85,B 0,C 180,E1 -20643.928,E2 -20643.928} C_VEL
LIN {X 0,Y 216.695,Z 637.16,A -85,B 0,C 180,E1 -20644.158,E2 -20644.158} C_VEL
LIN {X 0,Y 215.137,Z 629.547,A -85,B 0,C 180,E1 -20647.474,E2 -20647.474} C_VEL
LIN {X 0,Y 213.812,Z 623.855,A -85,B 0,C 180,E1 -20650.17,E2 -20650.17} C_VEL
LIN {X 0,Y 213.781,Z 623.858,A -85,B 0,C 180,E1 -20653.676,E2 -20653.676} C_VEL
LIN {X 0,Y 213.779,Z 623.858,A -85,B 0,C 180,E1 -20656.339,E2 -20656.339} C_VEL
LIN {X 0,Y 213.787,Z 623.855,A -85,B 0,C 180,E1 -20659.12,E2 -20659.12} C_VEL
LIN {X 0,Y 213.753,Z 623.859,A -85,B 0,C 180,E1 -20663.713,E2 -20663.713} C_VEL
LIN {X 0,Y 213.794,Z 623.853,A -85,B 0,C 180,E1 -20668.723,E2 -20668.723} C_VEL
LIN {X 0,Y 213.824,Z 623.85,A -85,B 0,C 180,E1 -20672.602,E2 -20672.602} C_VEL
LIN {X 0,Y 213.816,Z 623.852,A -85,B 0,C 180,E1 -20676.973,E2 -20676.973} C_VEL
LIN {X 0,Y 213.94,Z 623.831,A -85,B 0,C 180,E1 -20682.802,E2 -20682.802} C_VEL
LIN {X 0,Y 213.949,Z 623.835,A -85,B 0,C 180,E1 -20686.705,E2 -20686.705} C_VEL
LIN {X 0,Y 214.163,Z 623.797,A -85,B 0,C 180,E1 -20690.555,E2 -20690.555} C_VEL
LIN {X 0,Y 214.222,Z 623.795,A -85,B 0,C 180,E1 -20692.458,E2 -20692.458} C_VEL
LIN {X 0,Y 214.441,Z 623.768,A -85,B 0,C 180,E1 -20698.121,E2 -20698.121} C_VEL
LIN {X 0,Y 214.549,Z 623.748,A -85,B 0,C 180,E1 -20699.999,E2 -20699.999} C_VEL
LIN {X 0,Y 214.441,Z 623.763,A -85,B 0,C 180,E1 -20701.877,E2 -20701.877} C_VEL
LIN {X 0,Y 214.234,Z 623.8,A -85,B 0,C 180,E1 -20707.539,E2 -20707.539} C_VEL
LIN {X 0,Y 214.017,Z 623.817,A -85,B 0,C 180,E1 -20711.362,E2 -20711.362} C_VEL
LIN {X 0,Y 213.923,Z 623.827,A -85,B 0,C 180,E1 -20715.237,E2 -20715.237} C_VEL
LIN {X 0,Y 213.834,Z 623.846,A -85,B 0,C 180,E1 -20719.187,E2 -20719.187} C_VEL
LIN {X 0,Y 213.842,Z 623.84,A -85,B 0,C 180,E1 -20723.227,E2 -20723.227} C_VEL
LIN {X 0,Y 213.824,Z 623.838,A -85,B 0,C 180,E1 -20727.449,E2 -20727.449} C_VEL
LIN {X 0,Y 213.765,Z 623.856,A -85,B 0,C 180,E1 -20731.737,E2 -20731.737} C_VEL
LIN {X 0,Y 213.749,Z 623.849,A -85,B 0,C 180,E1 -20736.286,E2 -20736.286} C_VEL
LIN {X 0,Y 213.789,Z 623.849,A -85,B 0,C 180,E1 -20741.106,E2 -20741.106} C_VEL
LIN {X 0,Y 213.804,Z 623.851,A -85,B 0,C 180,E1 -20743.685,E2 -20743.685} C_VEL
LIN {X 0,Y 213.807,Z 623.85,A -85,B 0,C 180,E1 -20746.349,E2 -20746.349} C_VEL
LIN {X 0,Y 213.734,Z 623.854,A -85,B 0,C 180,E1 -20751.337,E2 -20751.337} C_VEL
LIN {X 0,Y 213.765,Z 623.857,A -85,B 0,C 180,E1 -20756.02,E2 -20756.02} C_VEL
LIN {X 0,Y 213.756,Z 623.851,A -85,B 0,C 180,E1 -20760.451,E2 -20760.451} C_VEL
LIN {X 0,Y 213.798,Z 623.853,A -85,B 0,C 180,E1 -20764.702,E2 -20764.702} C_VEL
LIN {X 0,Y 213.81,Z 623.851,A -85,B 0,C 180,E1 -20768.804,E2 -20768.804} C_VEL
LIN {X 0,Y 213.941,Z 623.835,A -85,B 0,C 180,E1 -20772.804,E2 -20772.804} C_VEL
LIN {X 0,Y 213.978,Z 623.829,A -85,B 0,C 180,E1 -20776.708,E2 -20776.708} C_VEL
LIN {X 0,Y 214.164,Z 623.805,A -85,B 0,C 180,E1 -20780.556,E2 -20780.556} C_VEL
LIN {X 0,Y 214.224,Z 623.796,A -85,B 0,C 180,E1 -20782.46,E2 -20782.46} C_VEL
LIN {X 0,Y 214.443,Z 623.769,A -85,B 0,C 180,E1 -20788.122,E2 -20788.122} C_VEL
LIN {X 0,Y 214.548,Z 623.756,A -85,B 0,C 180,E1 -20790,E2 -20790} C_VEL
LIN {X 0,Y 214.444,Z 623.77,A -85,B 0,C 180,E1 -20791.878,E2 -20791.878} C_VEL
LIN {X 0,Y 214.205,Z 623.803,A -85,B 0,C 180,E1 -20797.541,E2 -20797.541} C_VEL
LIN {X 0,Y 214.042,Z 623.824,A -85,B 0,C 180,E1 -20800.869,E2 -20800.869} C_VEL
LIN {X 0,Y 215.154,Z 626.871,A -85,B 0,C 180,E1 -20801.182,E2 -20801.182} C_VEL
LIN {X 0,Y 224.422,Z 647.136,A -85,B 0,C 180,E1 -20803.183,E2 -20803.183} C_VEL
LIN {X 0,Y 227.684,Z 655.454,A -85,B 0,C 180,E1 -20803.901,E2 -20803.901} C_VEL
LIN {X 0,Y 229.945,Z 661.864,A -85,B 0,C 180,E1 -20804.41,E2 -20804.41} C_VEL
LIN {X 0,Y 226.988,Z 725.717,A -85,B 0,C 180,E1 -20806.681,E2 -20806.681} C_VEL
LIN {X 0,Y 225.919,Z 739.809,A -85,B 0,C 180,E1 -20807.561,E2 -20807.561} C_VEL
LIN {X 0,Y 224.582,Z 751.886,A -85,B 0,C 180,E1 -20808.653,E2 -20808.653} C_VEL
LIN {X 0,Y 222.987,Z 763.588,A -85,B 0,C 180,E1 -20810.07,E2 -20810.07} C_VEL
LIN {X 0,Y 221.284,Z 773.992,A -85,B 0,C 180,E1 -20811.666,E2 -20811.666} C_VEL
LIN {X 0,Y 219.414,Z 784.134,A -85,B 0,C 180,E1 -20813.602,E2 -20813.602} C_VEL
LIN {X 0,Y 217.727,Z 793.014,A -85,B 0,C 180,E1 -20815.699,E2 -20815.699} C_VEL
LIN {X 0,Y 215.833,Z 802.345,A -85,B 0,C 180,E1 -20818.459,E2 -20818.459} C_VEL
LIN {X 0,Y 214.222,Z 810.379,A -85,B 0,C 180,E1 -20821.464,E2 -20821.464} C_VEL
LIN {X 0,Y 213.058,Z 816.555,A -85,B 0,C 180,E1 -20824.448,E2 -20824.448} C_VEL
LIN {X 0,Y 212.221,Z 821.23,A -85,B 0,C 180,E1 -20827.366,E2 -20827.366} C_VEL
LIN {X 0,Y 211.63,Z 824.652,A -85,B 0,C 180,E1 -20830.201,E2 -20830.201} C_VEL
LIN {X 0,Y 211.317,Z 827.034,A -85,B 0,C 180,E1 -20832.974,E2 -20832.974} C_VEL
LIN {X 0,Y 211.295,Z 828.507,A -85,B 0,C 180,E1 -20835.695,E2 -20835.695} C_VEL
LIN {X 0,Y 211.509,Z 829.119,A -85,B 0,C 180,E1 -20838.353,E2 -20838.353} C_VEL
LIN {X 0,Y 212.079,Z 828.96,A -85,B 0,C 180,E1 -20840.978,E2 -20840.978} C_VEL
LIN {X 0,Y 212.879,Z 828.086,A -85,B 0,C 180,E1 -20843.542,E2 -20843.542} C_VEL
LIN {X 0,Y 213.885,Z 826.491,A -85,B 0,C 180,E1 -20846.042,E2 -20846.042} C_VEL
LIN {X 0,Y 215.966,Z 822.736,A -85,B 0,C 180,E1 -20849.709,E2 -20849.709} C_VEL
LIN {X 0,Y 218.67,Z 817.325,A -85,B 0,C 180,E1 -20853.26,E2 -20853.26} C_VEL
LIN {X 0,Y 221.523,Z 811.167,A -85,B 0,C 180,E1 -20856.188,E2 -20856.188} C_VEL
LIN {X 0,Y 224.518,Z 804.389,A -85,B 0,C 180,E1 -20858.682,E2 -20858.682} C_VEL
LIN {X 0,Y 227.766,Z 796.152,A -85,B 0,C 180,E1 -20861.098,E2 -20861.098} C_VEL
LIN {X 0,Y 231.059,Z 787.089,A -85,B 0,C 180,E1 -20863.205,E2 -20863.205} C_VEL
LIN {X 0,Y 234.12,Z 777.39,A -85,B 0,C 180,E1 -20865.008,E2 -20865.008} C_VEL
LIN {X 0,Y 237.427,Z 765.281,A -85,B 0,C 180,E1 -20866.755,E2 -20866.755} C_VEL
LIN {X 0,Y 240.126,Z 753.047,A -85,B 0,C 180,E1 -20868.097,E2 -20868.097} C_VEL
LIN {X 0,Y 242.253,Z 739.384,A -85,B 0,C 180,E1 -20869.217,E2 -20869.217} C_VEL
LIN {X 0,Y 243.761,Z 726.381,A -85,B 0,C 180,E1 -20869.906,E2 -20869.906} C_VEL
LIN {X 0,Y 247.413,Z 675.707,A -85,B 0,C 180,E1 -20871.637,E2 -20871.637} C_VEL
LIN {X 0,Y 243.24,Z 666.526,A -85,B 0,C 180,E1 -20873.25,E2 -20873.25} C_VEL
LIN {X 0,Y 237.818,Z 656.368,A -85,B 0,C 180,E1 -20875.457,E2 -20875.457} C_VEL
LIN {X 0,Y 233.412,Z 649.373,A -85,B 0,C 180,E1 -20877.385,E2 -20877.385} C_VEL
LIN {X 0,Y 229.017,Z 643.059,A -85,B 0,C 180,E1 -20879.523,E2 -20879.523} C_VEL
LIN {X 0,Y 226.858,Z 639.73,A -85,B 0,C 180,E1 -20880.694,E2 -20880.694} C_VEL
LIN {X 0,Y 224.265,Z 636.621,A -85,B 0,C 180,E1 -20882.168,E2 -20882.168} C_VEL
LIN {X 0,Y 223.348,Z 635.206,A -85,B 0,C 180,E1 -20882.743,E2 -20882.743} C_VEL
LIN {X 0,Y 220.313,Z 632.561,A -85,B 0,C 180,E1 -20884.632,E2 -20884.632} C_VEL
LIN {X 0,Y 218.941,Z 630.262,A -85,B 0,C 180,E1 -20885.69,E2 -20885.69} C_VEL
LIN {X 0,Y 215.136,Z 626.571,A -85,B 0,C 180,E1 -20888.809,E2 -20888.809} C_VEL
LIN {X 0,Y 214.453,Z 625.138,A -85,B 0,C 180,E1 -20889.639,E2 -20889.639} C_VEL
LIN {X 0,Y 213.939,Z 623.831,A -85,B 0,C 180,E1 -20893.779,E2 -20893.779} C_VEL
LIN {X 0,Y 213.929,Z 623.838,A -85,B 0,C 180,E1 -20897.696,E2 -20897.696} C_VEL
LIN {X 0,Y 213.845,Z 623.84,A -85,B 0,C 180,E1 -20903.228,E2 -20903.228} C_VEL
LIN {X 0,Y 213.86,Z 624.198,A -85,B 0,C 180,E1 -20905.292,E2 -20905.292} C_VEL
LIN {X 0,Y 214.351,Z 625.955,A -85,B 0,C 180,E1 -20909.461,E2 -20909.461} C_VEL
LIN {X 0,Y 214.895,Z 627.216,A -85,B 0,C 180,E1 -20911.757,E2 -20911.757} C_VEL
LIN {X 0,Y 215.137,Z 628.069,A -85,B 0,C 180,E1 -20913.016,E2 -20913.016} C_VEL
LIN {X 0,Y 215.485,Z 629.878,A -85,B 0,C 180,E1 -20914.501,E2 -20914.501} C_VEL
LIN {X 0,Y 215.873,Z 632.795,A -85,B 0,C 180,E1 -20915.868,E2 -20915.868} C_VEL
LIN {X 0,Y 218.025,Z 642.397,A -85,B 0,C 180,E1 -20919.225,E2 -20919.225} C_VEL
LIN {X 0,Y 219.072,Z 644.503,A -85,B 0,C 180,E1 -20920.081,E2 -20920.081} C_VEL
LIN {X 0,Y 222.947,Z 650.64,A -85,B 0,C 180,E1 -20922.638,E2 -20922.638} C_VEL
LIN {X 0,Y 227.114,Z 657.669,A -85,B 0,C 180,E1 -20925.033,E2 -20925.033} C_VEL
LIN {X 0,Y 230.144,Z 663.215,A -85,B 0,C 180,E1 -20926.616,E2 -20926.616} C_VEL
LIN {X 0,Y 234.293,Z 671.328,A -85,B 0,C 180,E1 -20928.584,E2 -20928.584} C_VEL
LIN {X 0,Y 238.615,Z 681.342,A -85,B 0,C 180,E1 -20930.532,E2 -20930.532} C_VEL
LIN {X 0,Y 240.36,Z 686.21,A -85,B 0,C 180,E1 -20931.301,E2 -20931.301} C_VEL
LIN {X 0,Y 241.369,Z 698.812,A -85,B 0,C 180,E1 -20932.27,E2 -20932.27} C_VEL
LIN {X 0,Y 237.864,Z 743.732,A -85,B 0,C 180,E1 -20933.844,E2 -20933.844} C_VEL
LIN {X 0,Y 235.871,Z 757.688,A -85,B 0,C 180,E1 -20934.61,E2 -20934.61} C_VEL
LIN {X 0,Y 233.191,Z 770.388,A -85,B 0,C 180,E1 -20935.592,E2 -20935.592} C_VEL
LIN {X 0,Y 230.111,Z 782.496,A -85,B 0,C 180,E1 -20936.912,E2 -20936.912} C_VEL
LIN {X 0,Y 226.759,Z 793.503,A -85,B 0,C 180,E1 -20938.466,E2 -20938.466} C_VEL
LIN {X 0,Y 223.214,Z 803.57,A -85,B 0,C 180,E1 -20940.272,E2 -20940.272} C_VEL
LIN {X 0,Y 219.695,Z 812.715,A -85,B 0,C 180,E1 -20942.365,E2 -20942.365} C_VEL
LIN {X 0,Y 215.95,Z 821.702,A -85,B 0,C 180,E1 -20944.972,E2 -20944.972} C_VEL
LIN {X 0,Y 213.067,Z 828.484,A -85,B 0,C 180,E1 -20947.457,E2 -20947.457} C_VEL
LIN {X 0,Y 210.136,Z 834.983,A -85,B 0,C 180,E1 -20950.461,E2 -20950.461} C_VEL
LIN {X 0,Y 207.985,Z 839.711,A -85,B 0,C 180,E1 -20953.309,E2 -20953.309} C_VEL
LIN {X 0,Y 206.256,Z 843.361,A -85,B 0,C 180,E1 -20956.201,E2 -20956.201} C_VEL
LIN {X 0,Y 205.52,Z 845.239,A -85,B 0,C 180,E1 -20958.16,E2 -20958.16} C_VEL
LIN {X 0,Y 204.636,Z 847.775,A -85,B 0,C 180,E1 -20962.104,E2 -20962.104} C_VEL
LIN {X 0,Y 204.47,Z 848.668,A -85,B 0,C 180,E1 -20965.414,E2 -20965.414} C_VEL
LIN {X 0,Y 204.605,Z 848.563,A -85,B 0,C 180,E1 -20968.032,E2 -20968.032} C_VEL
LIN {X 0,Y 204.691,Z 848.002,A -85,B 0,C 180,E1 -20970,E2 -20970} C_VEL
LIN {X 0,Y 204.638,Z 847.022,A -85,B 0,C 180,E1 -20971.968,E2 -20971.968} C_VEL
LIN {X 0,Y 204.553,Z 844.73,A -85,B 0,C 180,E1 -20974.868,E2 -20974.868} C_VEL
LIN {X 0,Y 204.729,Z 841.278,A -85,B 0,C 180,E1 -20977.892,E2 -20977.892} C_VEL
LIN {X 0,Y 205.221,Z 836.736,A -85,B 0,C 180,E1 -20980.856,E2 -20980.856} C_VEL
LIN {X 0,Y 206.348,Z 829.78,A -85,B 0,C 180,E1 -20984.295,E2 -20984.295} C_VEL
LIN {X 0,Y 207.806,Z 822.183,A -85,B 0,C 180,E1 -20987.213,E2 -20987.213} C_VEL
LIN {X 0,Y 208.955,Z 816.053,A -85,B 0,C 180,E1 -20989.143,E2 -20989.143} C_VEL
LIN {X 0,Y 211.155,Z 805.996,A -85,B 0,C 180,E1 -20991.732,E2 -20991.732} C_VEL
LIN {X 0,Y 212.884,Z 796.988,A -85,B 0,C 180,E1 -20993.595,E2 -20993.595} C_VEL
LIN {X 0,Y 215.034,Z 785.989,A -85,B 0,C 180,E1 -20995.401,E2 -20995.401} C_VEL
LIN {X 0,Y 216.985,Z 773.729,A -85,B 0,C 180,E1 -20996.965,E2 -20996.965} C_VEL
LIN {X 0,Y 218.635,Z 760.948,A -85,B 0,C 180,E1 -20998.172,E2 -20998.172} C_VEL
LIN {X 0,Y 219.863,Z 748.543,A -85,B 0,C 180,E1 -20998.977,E2 -20998.977} C_VEL
LIN {X 0,Y 220.967,Z 727.914,A -85,B 0,C 180,E1 -20999.798,E2 -20999.798} C_VEL
LIN {X 0,Y 222.402,Z 693.385,A -85,B 0,C 180,E1 -21001.058,E2 -21001.058} C_VEL
LIN {X 0,Y 218.564,Z 661.691,A -85,B 0,C 180,E1 -21002.826,E2 -21002.826} C_VEL
LIN {X 0,Y 210.159,Z 639.111,A -85,B 0,C 180,E1 -21004.872,E2 -21004.872} C_VEL
LIN {X 0,Y 209.428,Z 636.759,A -85,B 0,C 180,E1 -21005.141,E2 -21005.141} C_VEL
LIN {X 0,Y 207.621,Z 628.64,A -85,B 0,C 180,E1 -21008.87,E2 -21008.87} C_VEL
LIN {X 0,Y 206.771,Z 624.734,A -85,B 0,C 180,E1 -21010.743,E2 -21010.743} C_VEL
LIN {X 0,Y 206.688,Z 624.74,A -85,B 0,C 180,E1 -21015.565,E2 -21015.565} C_VEL
LIN {X 0,Y 206.719,Z 624.734,A -85,B 0,C 180,E1 -21019.761,E2 -21019.761} C_VEL
LIN {X 0,Y 206.724,Z 624.734,A -85,B 0,C 180,E1 -21022.268,E2 -21022.268} C_VEL
LIN {X 0,Y 206.708,Z 624.738,A -85,B 0,C 180,E1 -21027.043,E2 -21027.043} C_VEL
LIN {X 0,Y 206.765,Z 624.728,A -85,B 0,C 180,E1 -21032.095,E2 -21032.095} C_VEL
LIN {X 0,Y 206.751,Z 624.73,A -85,B 0,C 180,E1 -21036.603,E2 -21036.603} C_VEL
LIN {X 0,Y 206.869,Z 624.709,A -85,B 0,C 180,E1 -21042.195,E2 -21042.195} C_VEL
LIN {X 0,Y 206.891,Z 624.713,A -85,B 0,C 180,E1 -21046.243,E2 -21046.243} C_VEL
LIN {X 0,Y 207.101,Z 624.676,A -85,B 0,C 180,E1 -21050.23,E2 -21050.23} C_VEL
LIN {X 0,Y 207.163,Z 624.674,A -85,B 0,C 180,E1 -21052.2,E2 -21052.2} C_VEL
LIN {X 0,Y 207.378,Z 624.648,A -85,B 0,C 180,E1 -21058.057,E2 -21058.057} C_VEL
LIN {X 0,Y 207.514,Z 624.624,A -85,B 0,C 180,E1 -21059.999,E2 -21059.999} C_VEL
LIN {X 0,Y 207.082,Z 624.687,A -85,B 0,C 180,E1 -21063.891,E2 -21063.891} C_VEL
LIN {X 0,Y 207.172,Z 624.678,A -85,B 0,C 180,E1 -21067.798,E2 -21067.798} C_VEL
LIN {X 0,Y 206.937,Z 624.695,A -85,B 0,C 180,E1 -21071.757,E2 -21071.757} C_VEL
LIN {X 0,Y 206.858,Z 624.71,A -85,B 0,C 180,E1 -21075.77,E2 -21075.77} C_VEL
LIN {X 0,Y 206.778,Z 624.727,A -85,B 0,C 180,E1 -21079.869,E2 -21079.869} C_VEL
LIN {X 0,Y 206.758,Z 624.716,A -85,B 0,C 180,E1 -21084.072,E2 -21084.072} C_VEL
LIN {X 0,Y 206.732,Z 624.728,A -85,B 0,C 180,E1 -21088.419,E2 -21088.419} C_VEL
LIN {X 0,Y 206.701,Z 624.734,A -85,B 0,C 180,E1 -21092.956,E2 -21092.956} C_VEL
LIN {X 0,Y 206.72,Z 624.72,A -85,B 0,C 180,E1 -21097.73,E2 -21097.73} C_VEL
LIN {X 0,Y 206.719,Z 624.731,A -85,B 0,C 180,E1 -21101.588,E2 -21101.588} C_VEL
LIN {X 0,Y 206.713,Z 624.734,A -85,B 0,C 180,E1 -21105.558,E2 -21105.558} C_VEL
LIN {X 0,Y 206.681,Z 624.726,A -85,B 0,C 180,E1 -21109.755,E2 -21109.755} C_VEL
LIN {X 0,Y 206.727,Z 624.735,A -85,B 0,C 180,E1 -21114.695,E2 -21114.695} C_VEL
LIN {X 0,Y 206.703,Z 624.726,A -85,B 0,C 180,E1 -21119.337,E2 -21119.337} C_VEL
LIN {X 0,Y 206.729,Z 624.733,A -85,B 0,C 180,E1 -21123.772,E2 -21123.772} C_VEL
LIN {X 0,Y 206.754,Z 624.73,A -85,B 0,C 180,E1 -21128.043,E2 -21128.043} C_VEL
LIN {X 0,Y 206.873,Z 624.714,A -85,B 0,C 180,E1 -21132.197,E2 -21132.197} C_VEL
LIN {X 0,Y 206.911,Z 624.708,A -85,B 0,C 180,E1 -21136.246,E2 -21136.246} C_VEL
LIN {X 0,Y 207.103,Z 624.683,A -85,B 0,C 180,E1 -21140.231,E2 -21140.231} C_VEL
LIN {X 0,Y 207.165,Z 624.675,A -85,B 0,C 180,E1 -21142.201,E2 -21142.201} C_VEL
LIN {X 0,Y 207.38,Z 624.649,A -85,B 0,C 180,E1 -21148.058,E2 -21148.058} C_VEL
LIN {X 0,Y 207.513,Z 624.633,A -85,B 0,C 180,E1 -21150,E2 -21150} C_VEL
LIN {X 0,Y 207.38,Z 624.65,A -85,B 0,C 180,E1 -21151.942,E2 -21151.942} C_VEL
LIN {X 0,Y 207.144,Z 624.682,A -85,B 0,C 180,E1 -21157.8,E2 -21157.8} C_VEL
LIN {X 0,Y 207.084,Z 624.69,A -85,B 0,C 180,E1 -21159.955,E2 -21159.955} C_VEL
LIN {X 0,Y 208.146,Z 627.645,A -85,B 0,C 180,E1 -21160.272,E2 -21160.272} C_VEL
LIN {X 0,Y 218.532,Z 650.444,A -85,B 0,C 180,E1 -21162.626,E2 -21162.626} C_VEL
LIN {X 0,Y 222.627,Z 661.032,A -85,B 0,C 180,E1 -21163.548,E2 -21163.548} C_VEL
LIN {X 0,Y 223.506,Z 663.589,A -85,B 0,C 180,E1 -21163.754,E2 -21163.754} C_VEL
LIN {X 0,Y 220.37,Z 726.344,A -85,B 0,C 180,E1 -21166.046,E2 -21166.046} C_VEL
LIN {X 0,Y 219.335,Z 739.413,A -85,B 0,C 180,E1 -21166.88,E2 -21166.88} C_VEL
LIN {X 0,Y 217.853,Z 752.48,A -85,B 0,C 180,E1 -21168.089,E2 -21168.089} C_VEL
LIN {X 0,Y 216.224,Z 763.887,A -85,B 0,C 180,E1 -21169.511,E2 -21169.511} C_VEL
LIN {X 0,Y 214.21,Z 775.618,A -85,B 0,C 180,E1 -21171.385,E2 -21171.385} C_VEL
LIN {X 0,Y 212.092,Z 786.803,A -85,B 0,C 180,E1 -21173.689,E2 -21173.689} C_VEL
LIN {X 0,Y 210.072,Z 796.86,A -85,B 0,C 180,E1 -21176.313,E2 -21176.313} C_VEL
LIN {X 0,Y 208.26,Z 805.315,A -85,B 0,C 180,E1 -21179.103,E2 -21179.103} C_VEL
LIN {X 0,Y 206.7,Z 813.073,A -85,B 0,C 180,E1 -21182.368,E2 -21182.368} C_VEL
LIN {X 0,Y 205.634,Z 818.858,A -85,B 0,C 180,E1 -21185.521,E2 -21185.521} C_VEL
LIN {X 0,Y 204.928,Z 822.555,A -85,B 0,C 180,E1 -21188.119,E2 -21188.119} C_VEL
LIN {X 0,Y 204.422,Z 825.527,A -85,B 0,C 180,E1 -21190.858,E2 -21190.858} C_VEL
LIN {X 0,Y 204.185,Z 827.719,A -85,B 0,C 180,E1 -21193.714,E2 -21193.714} C_VEL
LIN {X 0,Y 204.242,Z 829.024,A -85,B 0,C 180,E1 -21196.513,E2 -21196.513} C_VEL
LIN {X 0,Y 204.59,Z 829.529,A -85,B 0,C 180,E1 -21199.258,E2 -21199.258} C_VEL
LIN {X 0,Y 205.255,Z 829.229,A -85,B 0,C 180,E1 -21201.953,E2 -21201.953} C_VEL
LIN {X 0,Y 206.274,Z 828.066,A -85,B 0,C 180,E1 -21204.854,E2 -21204.854} C_VEL
LIN {X 0,Y 207.647,Z 825.963,A -85,B 0,C 180,E1 -21207.793,E2 -21207.793} C_VEL
LIN {X 0,Y 209.494,Z 822.841,A -85,B 0,C 180,E1 -21210.717,E2 -21210.717} C_VEL
LIN {X 0,Y 211.794,Z 818.573,A -85,B 0,C 180,E1 -21213.627,E2 -21213.627} C_VEL
LIN {X 0,Y 215.043,Z 812.1,A -85,B 0,C 180,E1 -21216.911,E2 -21216.911} C_VEL
LIN {X 0,Y 218.668,Z 804.414,A -85,B 0,C 180,E1 -21219.817,E2 -21219.817} C_VEL
LIN {X 0,Y 222.327,Z 795.691,A -85,B 0,C 180,E1 -21222.399,E2 -21222.399} C_VEL
LIN {X 0,Y 225.932,Z 785.942,A -85,B 0,C 180,E1 -21224.64,E2 -21224.64} C_VEL
LIN {X 0,Y 229.47,Z 775.217,A -85,B 0,C 180,E1 -21226.555,E2 -21226.555} C_VEL
LIN {X 0,Y 232.568,Z 764.012,A -85,B 0,C 180,E1 -21228.121,E2 -21228.121} C_VEL
LIN {X 0,Y 235.431,Z 751.061,A -85,B 0,C 180,E1 -21229.488,E2 -21229.488} C_VEL
LIN {X 0,Y 237.425,Z 738.378,A -85,B 0,C 180,E1 -21230.505,E2 -21230.505} C_VEL
LIN {X 0,Y 239.007,Z 724.698,A -85,B 0,C 180,E1 -21231.186,E2 -21231.186} C_VEL
LIN {X 0,Y 242.526,Z 678.356,A -85,B 0,C 180,E1 -21232.789,E2 -21232.789} C_VEL
LIN {X 0,Y 238.881,Z 670.389,A -85,B 0,C 180,E1 -21234.277,E2 -21234.277} C_VEL
LIN {X 0,Y 233.896,Z 660.796,A -85,B 0,C 180,E1 -21236.472,E2 -21236.472} C_VEL
LIN {X 0,Y 229.967,Z 654.473,A -85,B 0,C 180,E1 -21238.325,E2 -21238.325} C_VEL
LIN {X 0,Y 225.943,Z 648.499,A -85,B 0,C 180,E1 -21240.405,E2 -21240.405} C_VEL
LIN {X 0,Y 224.111,Z 645.691,A -85,B 0,C 180,E1 -21241.477,E2 -21241.477} C_VEL
LIN {X 0,Y 221.524,Z 642.195,A -85,B 0,C 180,E1 -21243.052,E2 -21243.052} C_VEL
LIN {X 0,Y 217.955,Z 638.534,A -85,B 0,C 180,E1 -21245.436,E2 -21245.436} C_VEL
LIN {X 0,Y 216.767,Z 636.607,A -85,B 0,C 180,E1 -21246.4,E2 -21246.4} C_VEL
LIN {X 0,Y 213.42,Z 633.19,A -85,B 0,C 180,E1 -21249.328,E2 -21249.328} C_VEL
LIN {X 0,Y 212.601,Z 631.8,A -85,B 0,C 180,E1 -21250.245,E2 -21250.245} C_VEL
LIN {X 0,Y 208.424,Z 628.331,A -85,B 0,C 180,E1 -21256.153,E2 -21256.153} C_VEL
LIN {X 0,Y 207.578,Z 627.145,A -85,B 0,C 180,E1 -21258.764,E2 -21258.764} C_VEL
LIN {X 0,Y 207.867,Z 627.73,A -85,B 0,C 180,E1 -21264.098,E2 -21264.098} C_VEL
LIN {X 0,Y 208.207,Z 629.216,A -85,B 0,C 180,E1 -21267.95,E2 -21267.95} C_VEL
LIN {X 0,Y 210.776,Z 633.435,A -85,B 0,C 180,E1 -21272.453,E2 -21272.453} C_VEL
LIN {X 0,Y 214.519,Z 637.963,A -85,B 0,C 180,E1 -21276.429,E2 -21276.429} C_VEL
LIN {X 0,Y 218.504,Z 643.856,A -85,B 0,C 180,E1 -21279.69,E2 -21279.69} C_VEL
LIN {X 0,Y 219.072,Z 644.503,A -85,B 0,C 180,E1 -21280.081,E2 -21280.081} C_VEL
LIN {X 0,Y 220.685,Z 647.864,A -85,B 0,C 180,E1 -21281.27,E2 -21281.27} C_VEL
LIN {X 0,Y 222.039,Z 651.989,A -85,B 0,C 180,E1 -21282.313,E2 -21282.313} C_VEL
LIN {X 0,Y 226.366,Z 667.251,A -85,B 0,C 180,E1 -21285.432,E2 -21285.432} C_VEL
LIN {X 0,Y 230.822,Z 676.522,A -85,B 0,C 180,E1 -21287.746,E2 -21287.746} C_VEL
LIN {X 0,Y 234.654,Z 685.808,A -85,B 0,C 180,E1 -21289.597,E2 -21289.597} C_VEL
LIN {X 0,Y 235.88,Z 689.313,A -85,B 0,C 180,E1 -21290.193,E2 -21290.193} C_VEL
LIN {X 0,Y 236.602,Z 700.299,A -85,B 0,C 180,E1 -21291.037,E2 -21291.037} C_VEL
LIN {X 0,Y 233.058,Z 743.606,A -85,B 0,C 180,E1 -21292.576,E2 -21292.576} C_VEL
LIN {X 0,Y 230.991,Z 757.361,A -85,B 0,C 180,E1 -21293.339,E2 -21293.339} C_VEL
LIN {X 0,Y 228.456,Z 768.993,A -85,B 0,C 180,E1 -21294.234,E2 -21294.234} C_VEL
LIN {X 0,Y 225.672,Z 779.716,A -85,B 0,C 180,E1 -21295.366,E2 -21295.366} C_VEL
LIN {X 0,Y 222.119,Z 791.082,A -85,B 0,C 180,E1 -21296.921,E2 -21296.921} C_VEL
LIN {X 0,Y 217.957,Z 802.558,A -85,B 0,C 180,E1 -21298.942,E2 -21298.942} C_VEL
LIN {X 0,Y 214.186,Z 811.842,A -85,B 0,C 180,E1 -21301.055,E2 -21301.055} C_VEL
LIN {X 0,Y 210.201,Z 820.914,A -85,B 0,C 180,E1 -21303.705,E2 -21303.705} C_VEL
LIN {X 0,Y 206.803,Z 828.205,A -85,B 0,C 180,E1 -21306.423,E2 -21306.423} C_VEL
LIN {X 0,Y 204.327,Z 833.346,A -85,B 0,C 180,E1 -21308.829,E2 -21308.829} C_VEL
LIN {X 0,Y 201.912,Z 838.329,A -85,B 0,C 180,E1 -21311.744,E2 -21311.744} C_VEL
LIN {X 0,Y 199.871,Z 842.221,A -85,B 0,C 180,E1 -21314.71,E2 -21314.71} C_VEL
LIN {X 0,Y 198.544,Z 845.115,A -85,B 0,C 180,E1 -21317.738,E2 -21317.738} C_VEL
LIN {X 0,Y 197.581,Z 847.542,A -85,B 0,C 180,E1 -21321.82,E2 -21321.82} C_VEL
LIN {X 0,Y 197.379,Z 848.352,A -85,B 0,C 180,E1 -21325.56,E2 -21325.56} C_VEL
LIN {X 0,Y 197.515,Z 848.141,A -85,B 0,C 180,E1 -21327.961,E2 -21327.961} C_VEL
LIN {X 0,Y 197.626,Z 847.536,A -85,B 0,C 180,E1 -21330,E2 -21330} C_VEL
LIN {X 0,Y 197.549,Z 846.486,A -85,B 0,C 180,E1 -21332.039,E2 -21332.039} C_VEL
LIN {X 0,Y 197.465,Z 844.37,A -85,B 0,C 180,E1 -21334.75,E2 -21334.75} C_VEL
LIN {X 0,Y 197.678,Z 840.547,A -85,B 0,C 180,E1 -21338.176,E2 -21338.176} C_VEL
LIN {X 0,Y 198.204,Z 835.874,A -85,B 0,C 180,E1 -21341.246,E2 -21341.246} C_VEL
LIN {X 0,Y 199.196,Z 829.89,A -85,B 0,C 180,E1 -21344.298,E2 -21344.298} C_VEL
LIN {X 0,Y 200.706,Z 822.395,A -85,B 0,C 180,E1 -21347.315,E2 -21347.315} C_VEL
LIN {X 0,Y 201.89,Z 816.377,A -85,B 0,C 180,E1 -21349.311,E2 -21349.311} C_VEL
LIN {X 0,Y 203.859,Z 807.433,A -85,B 0,C 180,E1 -21351.752,E2 -21351.752} C_VEL
LIN {X 0,Y 205.877,Z 797.606,A -85,B 0,C 180,E1 -21353.914,E2 -21353.914} C_VEL
LIN {X 0,Y 208.005,Z 786.904,A -85,B 0,C 180,E1 -21355.786,E2 -21355.786} C_VEL
LIN {X 0,Y 210.015,Z 774.985,A -85,B 0,C 180,E1 -21357.395,E2 -21357.395} C_VEL
LIN {X 0,Y 211.904,Z 761.536,A -85,B 0,C 180,E1 -21358.744,E2 -21358.744} C_VEL
LIN {X 0,Y 213.213,Z 748.563,A -85,B 0,C 180,E1 -21359.632,E2 -21359.632} C_VEL
LIN {X 0,Y 214.324,Z 729.042,A -85,B 0,C 180,E1 -21360.443,E2 -21360.443} C_VEL
LIN {X 0,Y 215.923,Z 694.877,A -85,B 0,C 180,E1 -21361.718,E2 -21361.718} C_VEL
LIN {X 0,Y 212.166,Z 663.606,A -85,B 0,C 180,E1 -21363.518,E2 -21363.518} C_VEL
LIN {X 0,Y 203.104,Z 639.208,A -85,B 0,C 180,E1 -21365.842,E2 -21365.842} C_VEL
LIN {X 0,Y 202.142,Z 636.449,A -85,B 0,C 180,E1 -21366.161,E2 -21366.161} C_VEL
LIN {X 0,Y 199.807,Z 626.204,A -85,B 0,C 180,E1 -21371.125,E2 -21371.125} C_VEL
LIN {X 0,Y 199.697,Z 625.613,A -85,B 0,C 180,E1 -21371.446,E2 -21371.446} C_VEL
LIN {X 0,Y 199.636,Z 625.62,A -85,B 0,C 180,E1 -21375.243,E2 -21375.243} C_VEL
LIN {X 0,Y 199.65,Z 625.616,A -85,B 0,C 180,E1 -21378.022,E2 -21378.022} C_VEL
LIN {X 0,Y 199.679,Z 625.613,A -85,B 0,C 180,E1 -21380.742,E2 -21380.742} C_VEL
LIN {X 0,Y 199.634,Z 625.618,A -85,B 0,C 180,E1 -21385.716,E2 -21385.716} C_VEL
LIN {X 0,Y 199.703,Z 625.608,A -85,B 0,C 180,E1 -21388.136,E2 -21388.136} C_VEL
LIN {X 0,Y 199.684,Z 625.61,A -85,B 0,C 180,E1 -21392.77,E2 -21392.77} C_VEL
LIN {X 0,Y 199.711,Z 625.61,A -85,B 0,C 180,E1 -21397.225,E2 -21397.225} C_VEL
LIN {X 0,Y 199.793,Z 625.591,A -85,B 0,C 180,E1 -21401.757,E2 -21401.757} C_VEL
LIN {X 0,Y 199.831,Z 625.594,A -85,B 0,C 180,E1 -21405.747,E2 -21405.747} C_VEL
LIN {X 0,Y 200.067,Z 625.553,A -85,B 0,C 180,E1 -21409.883,E2 -21409.883} C_VEL
LIN {X 0,Y 200.03,Z 625.567,A -85,B 0,C 180,E1 -21413.949,E2 -21413.949} C_VEL
LIN {X 0,Y 200.317,Z 625.528,A -85,B 0,C 180,E1 -21417.988,E2 -21417.988} C_VEL
LIN {X 0,Y 200.478,Z 625.5,A -85,B 0,C 180,E1 -21419.999,E2 -21419.999} C_VEL
LIN {X 0,Y 200.027,Z 625.565,A -85,B 0,C 180,E1 -21424.028,E2 -21424.028} C_VEL
LIN {X 0,Y 200.114,Z 625.556,A -85,B 0,C 180,E1 -21428.075,E2 -21428.075} C_VEL
LIN {X 0,Y 199.88,Z 625.571,A -85,B 0,C 180,E1 -21432.178,E2 -21432.178} C_VEL
LIN {X 0,Y 199.797,Z 625.592,A -85,B 0,C 180,E1 -21436.343,E2 -21436.343} C_VEL
LIN {X 0,Y 199.694,Z 625.606,A -85,B 0,C 180,E1 -21440.605,E2 -21440.605} C_VEL
LIN {X 0,Y 199.667,Z 625.596,A -85,B 0,C 180,E1 -21444.984,E2 -21444.984} C_VEL
LIN {X 0,Y 199.66,Z 625.609,A -85,B 0,C 180,E1 -21449.523,E2 -21449.523} C_VEL
LIN {X 0,Y 199.653,Z 625.614,A -85,B 0,C 180,E1 -21452.349,E2 -21452.349} C_VEL
LIN {X 0,Y 199.648,Z 625.602,A -85,B 0,C 180,E1 -21456.756,E2 -21456.756} C_VEL
LIN {X 0,Y 199.674,Z 625.6,A -85,B 0,C 180,E1 -21459.311,E2 -21459.311} C_VEL
LIN {X 0,Y 199.658,Z 625.614,A -85,B 0,C 180,E1 -21462.338,E2 -21462.338} C_VEL
LIN {X 0,Y 199.661,Z 625.612,A -85,B 0,C 180,E1 -21465.253,E2 -21465.253} C_VEL
LIN {X 0,Y 199.637,Z 625.609,A -85,B 0,C 180,E1 -21468.021,E2 -21468.021} C_VEL
LIN {X 0,Y 199.639,Z 625.608,A -85,B 0,C 180,E1 -21470.756,E2 -21470.756} C_VEL
LIN {X 0,Y 199.629,Z 625.617,A -85,B 0,C 180,E1 -21475.718,E2 -21475.718} C_VEL
LIN {X 0,Y 199.692,Z 625.605,A -85,B 0,C 180,E1 -21478.136,E2 -21478.136} C_VEL
LIN {X 0,Y 199.682,Z 625.613,A -85,B 0,C 180,E1 -21482.772,E2 -21482.772} C_VEL
LIN {X 0,Y 199.735,Z 625.604,A -85,B 0,C 180,E1 -21487.229,E2 -21487.229} C_VEL
LIN {X 0,Y 199.834,Z 625.591,A -85,B 0,C 180,E1 -21491.722,E2 -21491.722} C_VEL
LIN {X 0,Y 199.845,Z 625.587,A -85,B 0,C 180,E1 -21495.749,E2 -21495.749} C_VEL
LIN {X 0,Y 200.067,Z 625.559,A -85,B 0,C 180,E1 -21499.884,E2 -21499.884} C_VEL
LIN {X 0,Y 200.032,Z 625.564,A -85,B 0,C 180,E1 -21503.95,E2 -21503.95} C_VEL
LIN {X 0,Y 200.32,Z 625.529,A -85,B 0,C 180,E1 -21507.989,E2 -21507.989} C_VEL
LIN {X 0,Y 200.477,Z 625.509,A -85,B 0,C 180,E1 -21510,E2 -21510} C_VEL
LIN {X 0,Y 200.028,Z 625.566,A -85,B 0,C 180,E1 -21514.029,E2 -21514.029} C_VEL
LIN {X 0,Y 200.05,Z 625.567,A -85,B 0,C 180,E1 -21518.968,E2 -21518.968} C_VEL
LIN {X 0,Y 201.206,Z 628.651,A -85,B 0,C 180,E1 -21519.328,E2 -21519.328} C_VEL
LIN {X 0,Y 211.889,Z 651.986,A -85,B 0,C 180,E1 -21521.864,E2 -21521.864} C_VEL
LIN {X 0,Y 215.644,Z 661.433,A -85,B 0,C 180,E1 -21522.745,E2 -21522.745} C_VEL
LIN {X 0,Y 216.942,Z 665.205,A -85,B 0,C 180,E1 -21523.062,E2 -21523.062} C_VEL
LIN {X 0,Y 213.789,Z 726.062,A -85,B 0,C 180,E1 -21525.344,E2 -21525.344} C_VEL
LIN {X 0,Y 212.661,Z 739.949,A -85,B 0,C 180,E1 -21526.252,E2 -21526.252} C_VEL
LIN {X 0,Y 211.203,Z 752.362,A -85,B 0,C 180,E1 -21527.426,E2 -21527.426} C_VEL
LIN {X 0,Y 209.311,Z 765.341,A -85,B 0,C 180,E1 -21529.109,E2 -21529.109} C_VEL
LIN {X 0,Y 207.405,Z 775.791,A -85,B 0,C 180,E1 -21530.842,E2 -21530.842} C_VEL
LIN {X 0,Y 205.442,Z 785.95,A -85,B 0,C 180,E1 -21532.959,E2 -21532.959} C_VEL
LIN {X 0,Y 203.429,Z 795.629,A -85,B 0,C 180,E1 -21535.493,E2 -21535.493} C_VEL
LIN {X 0,Y 201.377,Z 805.03,A -85,B 0,C 180,E1 -21538.591,E2 -21538.591} C_VEL
LIN {X 0,Y 199.788,Z 812.659,A -85,B 0,C 180,E1 -21541.847,E2 -21541.847} C_VEL
LIN {X 0,Y 198.831,Z 817.514,A -85,B 0,C 180,E1 -21544.439,E2 -21544.439} C_VEL
LIN {X 0,Y 198.07,Z 821.543,A -85,B 0,C 180,E1 -21547.098,E2 -21547.098} C_VEL
LIN {X 0,Y 197.474,Z 824.786,A -85,B 0,C 180,E1 -21549.836,E2 -21549.836} C_VEL
LIN {X 0,Y 197.143,Z 827.211,A -85,B 0,C 180,E1 -21552.634,E2 -21552.634} C_VEL
LIN {X 0,Y 197.076,Z 828.87,A -85,B 0,C 180,E1 -21555.497,E2 -21555.497} C_VEL
LIN {X 0,Y 197.331,Z 829.752,A -85,B 0,C 180,E1 -21558.409,E2 -21558.409} C_VEL
LIN {X 0,Y 197.967,Z 829.825,A -85,B 0,C 180,E1 -21561.352,E2 -21561.352} C_VEL
LIN {X 0,Y 198.958,Z 829.02,A -85,B 0,C 180,E1 -21564.334,E2 -21564.334} C_VEL
LIN {X 0,Y 200.805,Z 826.525,A -85,B 0,C 180,E1 -21568.334,E2 -21568.334} C_VEL
LIN {X 0,Y 202.47,Z 823.993,A -85,B 0,C 180,E1 -21570.926,E2 -21570.926} C_VEL
LIN {X 0,Y 205.536,Z 818.742,A -85,B 0,C 180,E1 -21574.697,E2 -21574.697} C_VEL
LIN {X 0,Y 208.829,Z 812.709,A -85,B 0,C 180,E1 -21577.842,E2 -21577.842} C_VEL
LIN {X 0,Y 212.469,Z 805.464,A -85,B 0,C 180,E1 -21580.685,E2 -21580.685} C_VEL
LIN {X 0,Y 215.72,Z 798.217,A -85,B 0,C 180,E1 -21582.951,E2 -21582.951} C_VEL
LIN {X 0,Y 219.762,Z 788.228,A -85,B 0,C 180,E1 -21585.414,E2 -21585.414} C_VEL
LIN {X 0,Y 223.312,Z 778.328,A -85,B 0,C 180,E1 -21587.316,E2 -21587.316} C_VEL
LIN {X 0,Y 226.85,Z 766.659,A -85,B 0,C 180,E1 -21589.062,E2 -21589.062} C_VEL
LIN {X 0,Y 229.844,Z 754.604,A -85,B 0,C 180,E1 -21590.441,E2 -21590.441} C_VEL
LIN {X 0,Y 232.224,Z 741.103,A -85,B 0,C 180,E1 -21591.599,E2 -21591.599} C_VEL
LIN {X 0,Y 233.998,Z 727.558,A -85,B 0,C 180,E1 -21592.354,E2 -21592.354} C_VEL
LIN {X 0,Y 237.784,Z 681.148,A -85,B 0,C 180,E1 -21593.97,E2 -21593.97} C_VEL
LIN {X 0,Y 233.648,Z 672.182,A -85,B 0,C 180,E1 -21595.83,E2 -21595.83} C_VEL
LIN {X 0,Y 229.506,Z 664.204,A -85,B 0,C 180,E1 -21597.818,E2 -21597.818} C_VEL
LIN {X 0,Y 226.425,Z 659.369,A -85,B 0,C 180,E1 -21599.379,E2 -21599.379} C_VEL
LIN {X 0,Y 221.837,Z 652.045,A -85,B 0,C 180,E1 -21602.035,E2 -21602.035} C_VEL
LIN {X 0,Y 218.719,Z 647.959,A -85,B 0,C 180,E1 -21604.032,E2 -21604.032} C_VEL
LIN {X 0,Y 215.907,Z 644.948,A -85,B 0,C 180,E1 -21606.044,E2 -21606.044} C_VEL
LIN {X 0,Y 214.413,Z 642.629,A -85,B 0,C 180,E1 -21607.328,E2 -21607.328} C_VEL
LIN {X 0,Y 211.77,Z 639.882,A -85,B 0,C 180,E1 -21609.803,E2 -21609.803} C_VEL
LIN {X 0,Y 210.97,Z 638.561,A -85,B 0,C 180,E1 -21610.726,E2 -21610.726} C_VEL
LIN {X 0,Y 207.065,Z 635.101,A -85,B 0,C 180,E1 -21616.722,E2 -21616.722} C_VEL
LIN {X 0,Y 206.374,Z 634.14,A -85,B 0,C 180,E1 -21618.985,E2 -21618.985} C_VEL
LIN {X 0,Y 206.061,Z 634.645,A -85,B 0,C 180,E1 -21624.16,E2 -21624.16} C_VEL
LIN {X 0,Y 206.97,Z 636.135,A -85,B 0,C 180,E1 -21627.667,E2 -21627.667} C_VEL
LIN {X 0,Y 209.605,Z 640.619,A -85,B 0,C 180,E1 -21632.445,E2 -21632.445} C_VEL
LIN {X 0,Y 212.731,Z 644.559,A -85,B 0,C 180,E1 -21635.892,E2 -21635.892} C_VEL
LIN {X 0,Y 216.552,Z 650.414,A -85,B 0,C 180,E1 -21639.191,E2 -21639.191} C_VEL
LIN {X 0,Y 221.1,Z 657.977,A -85,B 0,C 180,E1 -21642.367,E2 -21642.367} C_VEL
LIN {X 0,Y 224.42,Z 663.811,A -85,B 0,C 180,E1 -21644.374,E2 -21644.374} C_VEL
LIN {X 0,Y 226.366,Z 667.251,A -85,B 0,C 180,E1 -21645.432,E2 -21645.432} C_VEL
LIN {X 0,Y 228.787,Z 674.932,A -85,B 0,C 180,E1 -21646.904,E2 -21646.904} C_VEL
LIN {X 0,Y 229.89,Z 680.014,A -85,B 0,C 180,E1 -21647.644,E2 -21647.644} C_VEL
LIN {X 0,Y 231.409,Z 690.881,A -85,B 0,C 180,E1 -21648.865,E2 -21648.865} C_VEL
LIN {X 0,Y 231.736,Z 694.632,A -85,B 0,C 180,E1 -21649.209,E2 -21649.209} C_VEL
LIN {X 0,Y 232.082,Z 700.916,A -85,B 0,C 180,E1 -21649.712,E2 -21649.712} C_VEL
LIN {X 0,Y 228.366,Z 743.423,A -85,B 0,C 180,E1 -21651.249,E2 -21651.249} C_VEL
LIN {X 0,Y 226.191,Z 757.11,A -85,B 0,C 180,E1 -21652.006,E2 -21652.006} C_VEL
LIN {X 0,Y 223.34,Z 769.659,A -85,B 0,C 180,E1 -21653.001,E2 -21653.001} C_VEL
LIN {X 0,Y 219.964,Z 781.7,A -85,B 0,C 180,E1 -21654.332,E2 -21654.332} C_VEL
LIN {X 0,Y 216.3,Z 792.657,A -85,B 0,C 180,E1 -21655.912,E2 -21655.912} C_VEL
LIN {X 0,Y 212.38,Z 802.699,A -85,B 0,C 180,E1 -21657.752,E2 -21657.752} C_VEL
LIN {X 0,Y 208.054,Z 812.638,A -85,B 0,C 180,E1 -21660.116,E2 -21660.116} C_VEL
LIN {X 0,Y 203.904,Z 821.497,A -85,B 0,C 180,E1 -21662.827,E2 -21662.827} C_VEL
LIN {X 0,Y 200.25,Z 828.794,A -85,B 0,C 180,E1 -21665.692,E2 -21665.692} C_VEL
LIN {X 0,Y 196.775,Z 835.354,A -85,B 0,C 180,E1 -21669.075,E2 -21669.075} C_VEL
LIN {X 0,Y 194.382,Z 839.816,A -85,B 0,C 180,E1 -21672.103,E2 -21672.103} C_VEL
LIN {X 0,Y 192.425,Z 843.241,A -85,B 0,C 180,E1 -21675.187,E2 -21675.187} C_VEL
LIN {X 0,Y 190.958,Z 846.351,A -85,B 0,C 180,E1 -21679.396,E2 -21679.396} C_VEL
LIN {X 0,Y 190.527,Z 847.299,A -85,B 0,C 180,E1 -21681.515,E2 -21681.515} C_VEL
LIN {X 0,Y 190.319,Z 847.964,A -85,B 0,C 180,E1 -21685.765,E2 -21685.765} C_VEL
LIN {X 0,Y 190.427,Z 847.714,A -85,B 0,C 180,E1 -21687.885,E2 -21687.885} C_VEL
LIN {X 0,Y 190.56,Z 847.058,A -85,B 0,C 180,E1 -21690,E2 -21690} C_VEL
LIN {X 0,Y 190.463,Z 845.918,A -85,B 0,C 180,E1 -21692.115,E2 -21692.115} C_VEL
LIN {X 0,Y 190.402,Z 843.938,A -85,B 0,C 180,E1 -21694.71,E2 -21694.71} C_VEL
LIN {X 0,Y 190.647,Z 839.777,A -85,B 0,C 180,E1 -21698.479,E2 -21698.479} C_VEL
LIN {X 0,Y 191.209,Z 834.978,A -85,B 0,C 180,E1 -21701.663,E2 -21701.663} C_VEL
LIN {X 0,Y 192.295,Z 828.865,A -85,B 0,C 180,E1 -21704.823,E2 -21704.823} C_VEL
LIN {X 0,Y 193.887,Z 821.22,A -85,B 0,C 180,E1 -21707.945,E2 -21707.945} C_VEL
LIN {X 0,Y 195.579,Z 812.805,A -85,B 0,C 180,E1 -21710.685,E2 -21710.685} C_VEL
LIN {X 0,Y 197.697,Z 803.824,A -85,B 0,C 180,E1 -21713.019,E2 -21713.019} C_VEL
LIN {X 0,Y 199.895,Z 793.219,A -85,B 0,C 180,E1 -21715.232,E2 -21715.232} C_VEL
LIN {X 0,Y 202.148,Z 781.476,A -85,B 0,C 180,E1 -21717.149,E2 -21717.149} C_VEL
LIN {X 0,Y 204.178,Z 769.065,A -85,B 0,C 180,E1 -21718.668,E2 -21718.668} C_VEL
LIN {X 0,Y 205.967,Z 755.558,A -85,B 0,C 180,E1 -21719.865,E2 -21719.865} C_VEL
LIN {X 0,Y 207.082,Z 741.846,A -85,B 0,C 180,E1 -21720.655,E2 -21720.655} C_VEL
LIN {X 0,Y 209.317,Z 695.151,A -85,B 0,C 180,E1 -21722.472,E2 -21722.472} C_VEL
LIN {X 0,Y 205.866,Z 665.579,A -85,B 0,C 180,E1 -21724.241,E2 -21724.241} C_VEL
LIN {X 0,Y 196.186,Z 639.688,A -85,B 0,C 180,E1 -21726.828,E2 -21726.828} C_VEL
LIN {X 0,Y 194.828,Z 636.118,A -85,B 0,C 180,E1 -21727.262,E2 -21727.262} C_VEL
LIN {X 0,Y 193.18,Z 628.849,A -85,B 0,C 180,E1 -21730.907,E2 -21730.907} C_VEL
LIN {X 0,Y 192.613,Z 626.497,A -85,B 0,C 180,E1 -21732.161,E2 -21732.161} C_VEL
LIN {X 0,Y 192.566,Z 626.499,A -85,B 0,C 180,E1 -21736.879,E2 -21736.879} C_VEL
LIN {X 0,Y 192.599,Z 626.493,A -85,B 0,C 180,E1 -21741.658,E2 -21741.658} C_VEL
LIN {X 0,Y 192.599,Z 626.497,A -85,B 0,C 180,E1 -21746.813,E2 -21746.813} C_VEL
LIN {X 0,Y 192.663,Z 626.485,A -85,B 0,C 180,E1 -21751.691,E2 -21751.691} C_VEL
LIN {X 0,Y 192.683,Z 626.482,A -85,B 0,C 180,E1 -21756.344,E2 -21756.344} C_VEL
LIN {X 0,Y 192.728,Z 626.47,A -85,B 0,C 180,E1 -21761.458,E2 -21761.458} C_VEL
LIN {X 0,Y 192.76,Z 626.477,A -85,B 0,C 180,E1 -21765.212,E2 -21765.212} C_VEL
LIN {X 0,Y 192.978,Z 626.437,A -85,B 0,C 180,E1 -21769.507,E2 -21769.507} C_VEL
LIN {X 0,Y 193.057,Z 626.429,A -85,B 0,C 180,E1 -21771.626,E2 -21771.626} C_VEL
LIN {X 0,Y 193.259,Z 626.407,A -85,B 0,C 180,E1 -21777.915,E2 -21777.915} C_VEL
LIN {X 0,Y 193.441,Z 626.376,A -85,B 0,C 180,E1 -21779.999,E2 -21779.999} C_VEL
LIN {X 0,Y 192.974,Z 626.443,A -85,B 0,C 180,E1 -21784.176,E2 -21784.176} C_VEL
LIN {X 0,Y 193.063,Z 626.433,A -85,B 0,C 180,E1 -21788.372,E2 -21788.372} C_VEL
LIN {X 0,Y 192.803,Z 626.45,A -85,B 0,C 180,E1 -21792.632,E2 -21792.632} C_VEL
LIN {X 0,Y 192.751,Z 626.469,A -85,B 0,C 180,E1 -21796.958,E2 -21796.958} C_VEL
LIN {X 0,Y 192.631,Z 626.487,A -85,B 0,C 180,E1 -21801.397,E2 -21801.397} C_VEL
LIN {X 0,Y 192.659,Z 626.47,A -85,B 0,C 180,E1 -21804.224,E2 -21804.224} C_VEL
LIN {X 0,Y 192.639,Z 626.482,A -85,B 0,C 180,E1 -21808.888,E2 -21808.888} C_VEL
LIN {X 0,Y 192.593,Z 626.491,A -85,B 0,C 180,E1 -21813.185,E2 -21813.185} C_VEL
LIN {X 0,Y 192.595,Z 626.478,A -85,B 0,C 180,E1 -21818.34,E2 -21818.34} C_VEL
LIN {X 0,Y 192.6,Z 626.492,A -85,B 0,C 180,E1 -21823.132,E2 -21823.132} C_VEL
LIN {X 0,Y 192.589,Z 626.489,A -85,B 0,C 180,E1 -21826.872,E2 -21826.872} C_VEL
LIN {X 0,Y 192.571,Z 626.49,A -85,B 0,C 180,E1 -21831.654,E2 -21831.654} C_VEL
LIN {X 0,Y 192.594,Z 626.495,A -85,B 0,C 180,E1 -21834.279,E2 -21834.279} C_VEL
LIN {X 0,Y 192.596,Z 626.482,A -85,B 0,C 180,E1 -21839.279,E2 -21839.279} C_VEL
LIN {X 0,Y 192.657,Z 626.483,A -85,B 0,C 180,E1 -21841.691,E2 -21841.691} C_VEL
LIN {X 0,Y 192.702,Z 626.479,A -85,B 0,C 180,E1 -21846.349,E2 -21846.349} C_VEL
LIN {X 0,Y 192.778,Z 626.47,A -85,B 0,C 180,E1 -21851.414,E2 -21851.414} C_VEL
LIN {X 0,Y 192.85,Z 626.46,A -85,B 0,C 180,E1 -21857.37,E2 -21857.37} C_VEL
LIN {X 0,Y 193.059,Z 626.432,A -85,B 0,C 180,E1 -21861.627,E2 -21861.627} C_VEL
LIN {X 0,Y 193.262,Z 626.408,A -85,B 0,C 180,E1 -21867.916,E2 -21867.916} C_VEL
LIN {X 0,Y 193.441,Z 626.386,A -85,B 0,C 180,E1 -21870,E2 -21870} C_VEL
LIN {X 0,Y 192.974,Z 626.445,A -85,B 0,C 180,E1 -21874.177,E2 -21874.177} C_VEL
LIN {X 0,Y 193.038,Z 626.465,A -85,B 0,C 180,E1 -21877.978,E2 -21877.978} C_VEL
LIN {X 0,Y 194.114,Z 629.411,A -85,B 0,C 180,E1 -21878.294,E2 -21878.294} C_VEL
LIN {X 0,Y 205.459,Z 653.791,A -85,B 0,C 180,E1 -21881.093,E2 -21881.093} C_VEL
LIN {X 0,Y 209.709,Z 664.654,A -85,B 0,C 180,E1 -21882.147,E2 -21882.147} C_VEL
LIN {X 0,Y 210.361,Z 667.323,A -85,B 0,C 180,E1 -21882.349,E2 -21882.349} C_VEL
LIN {X 0,Y 207.17,Z 727.143,A -85,B 0,C 180,E1 -21884.677,E2 -21884.677} C_VEL
LIN {X 0,Y 206,Z 740.517,A -85,B 0,C 180,E1 -21885.585,E2 -21885.585} C_VEL
LIN {X 0,Y 204.469,Z 753.035,A -85,B 0,C 180,E1 -21886.814,E2 -21886.814} C_VEL
LIN {X 0,Y 202.656,Z 765.098,A -85,B 0,C 180,E1 -21888.419,E2 -21888.419} C_VEL
LIN {X 0,Y 200.61,Z 775.994,A -85,B 0,C 180,E1 -21890.266,E2 -21890.266} C_VEL
LIN {X 0,Y 198.714,Z 785.522,A -85,B 0,C 180,E1 -21892.292,E2 -21892.292} C_VEL
LIN {X 0,Y 196.696,Z 795.074,A -85,B 0,C 180,E1 -21894.823,E2 -21894.823} C_VEL
LIN {X 0,Y 194.851,Z 803.236,A -85,B 0,C 180,E1 -21897.504,E2 -21897.504} C_VEL
LIN {X 0,Y 193.169,Z 810.833,A -85,B 0,C 180,E1 -21900.62,E2 -21900.62} C_VEL
LIN {X 0,Y 191.871,Z 817.211,A -85,B 0,C 180,E1 -21903.957,E2 -21903.957} C_VEL
LIN {X 0,Y 190.867,Z 822.244,A -85,B 0,C 180,E1 -21907.41,E2 -21907.41} C_VEL
LIN {X 0,Y 190.286,Z 825.524,A -85,B 0,C 180,E1 -21910.384,E2 -21910.384} C_VEL
LIN {X 0,Y 190.065,Z 827.148,A -85,B 0,C 180,E1 -21912.31,E2 -21912.31} C_VEL
LIN {X 0,Y 189.974,Z 829.016,A -85,B 0,C 180,E1 -21915.342,E2 -21915.342} C_VEL
LIN {X 0,Y 190.221,Z 830.035,A -85,B 0,C 180,E1 -21918.316,E2 -21918.316} C_VEL
LIN {X 0,Y 190.837,Z 830.233,A -85,B 0,C 180,E1 -21921.241,E2 -21921.241} C_VEL
LIN {X 0,Y 191.734,Z 829.704,A -85,B 0,C 180,E1 -21924.094,E2 -21924.094} C_VEL
LIN {X 0,Y 192.939,Z 828.473,A -85,B 0,C 180,E1 -21926.906,E2 -21926.906} C_VEL
LIN {X 0,Y 195.45,Z 825.087,A -85,B 0,C 180,E1 -21931.151,E2 -21931.151} C_VEL
LIN {X 0,Y 197.667,Z 821.694,A -85,B 0,C 180,E1 -21933.998,E2 -21933.998} C_VEL
LIN {X 0,Y 200.98,Z 816.24,A -85,B 0,C 180,E1 -21937.379,E2 -21937.379} C_VEL
LIN {X 0,Y 204.7,Z 809.572,A -85,B 0,C 180,E1 -21940.444,E2 -21940.444} C_VEL
LIN {X 0,Y 208.89,Z 801.227,A -85,B 0,C 180,E1 -21943.384,E2 -21943.384} C_VEL
LIN {X 0,Y 212.613,Z 793.009,A -85,B 0,C 180,E1 -21945.647,E2 -21945.647} C_VEL
LIN {X 0,Y 216.404,Z 783.458,A -85,B 0,C 180,E1 -21947.74,E2 -21947.74} C_VEL
LIN {X 0,Y 220.231,Z 772.466,A -85,B 0,C 180,E1 -21949.59,E2 -21949.59} C_VEL
LIN {X 0,Y 223.683,Z 760.3,A -85,B 0,C 180,E1 -21951.188,E2 -21951.188} C_VEL
LIN {X 0,Y 226.473,Z 747.722,A -85,B 0,C 180,E1 -21952.41,E2 -21952.41} C_VEL
LIN {X 0,Y 228.36,Z 735.924,A -85,B 0,C 180,E1 -21953.274,E2 -21953.274} C_VEL
LIN {X 0,Y 229.873,Z 723.03,A -85,B 0,C 180,E1 -21953.867,E2 -21953.867} C_VEL
LIN {X 0,Y 233.156,Z 683.87,A -85,B 0,C 180,E1 -21955.251,E2 -21955.251} C_VEL
LIN {X 0,Y 228.236,Z 673.234,A -85,B 0,C 180,E1 -21957.663,E2 -21957.663} C_VEL
LIN {X 0,Y 224.627,Z 666.695,A -85,B 0,C 180,E1 -21959.575,E2 -21959.575} C_VEL
LIN {X 0,Y 219.268,Z 658.078,A -85,B 0,C 180,E1 -21962.794,E2 -21962.794} C_VEL
LIN {X 0,Y 216.561,Z 654.4,A -85,B 0,C 180,E1 -21964.649,E2 -21964.649} C_VEL
LIN {X 0,Y 213.723,Z 651.051,A -85,B 0,C 180,E1 -21966.817,E2 -21966.817} C_VEL
LIN {X 0,Y 212.623,Z 649.27,A -85,B 0,C 180,E1 -21967.838,E2 -21967.838} C_VEL
LIN {X 0,Y 210.066,Z 646.425,A -85,B 0,C 180,E1 -21970.37,E2 -21970.37} C_VEL
LIN {X 0,Y 209.391,Z 645.339,A -85,B 0,C 180,E1 -21971.213,E2 -21971.213} C_VEL
LIN {X 0,Y 206.01,Z 642.233,A -85,B 0,C 180,E1 -21976.567,E2 -21976.567} C_VEL
LIN {X 0,Y 205.242,Z 641.146,A -85,B 0,C 180,E1 -21979.094,E2 -21979.094} C_VEL
LIN {X 0,Y 204.912,Z 641.559,A -85,B 0,C 180,E1 -21983.782,E2 -21983.782} C_VEL
LIN {X 0,Y 205.774,Z 643.15,A -85,B 0,C 180,E1 -21987.489,E2 -21987.489} C_VEL
LIN {X 0,Y 207.925,Z 647.101,A -85,B 0,C 180,E1 -21991.728,E2 -21991.728} C_VEL
LIN {X 0,Y 210.912,Z 651.046,A -85,B 0,C 180,E1 -21995.28,E2 -21995.28} C_VEL
LIN {X 0,Y 214.417,Z 656.715,A -85,B 0,C 180,E1 -21998.52,E2 -21998.52} C_VEL
LIN {X 0,Y 218.547,Z 663.971,A -85,B 0,C 180,E1 -22001.611,E2 -22001.611} C_VEL
LIN {X 0,Y 221.574,Z 669.502,A -85,B 0,C 180,E1 -22003.562,E2 -22003.562} C_VEL
LIN {X 0,Y 224.41,Z 675.153,A -85,B 0,C 180,E1 -22005.219,E2 -22005.219} C_VEL
LIN {X 0,Y 228.095,Z 683.328,A -85,B 0,C 180,E1 -22007.242,E2 -22007.242} C_VEL
LIN {X 0,Y 231.577,Z 692.512,A -85,B 0,C 180,E1 -22009.024,E2 -22009.024} C_VEL
LIN {X 0,Y 231.736,Z 694.632,A -85,B 0,C 180,E1 -22009.209,E2 -22009.209} C_VEL
LIN {X 0,Y 231.569,Z 697.826,A -85,B 0,C 180,E1 -22009.354,E2 -22009.354} C_VEL
LIN {X 0,Y 230.424,Z 702.321,A -85,B 0,C 180,E1 -22009.264,E2 -22009.264} C_VEL
LIN {X 0,Y 227.294,Z 711.223,A -85,B 0,C 180,E1 -22008.8,E2 -22008.8} C_VEL
LIN {X 0,Y 226.554,Z 715.231,A -85,B 0,C 180,E1 -22008.812,E2 -22008.812} C_VEL
LIN {X 0,Y 223.883,Z 743.503,A -85,B 0,C 180,E1 -22009.855,E2 -22009.855} C_VEL
LIN {X 0,Y 221.563,Z 757.216,A -85,B 0,C 180,E1 -22010.626,E2 -22010.626} C_VEL
LIN {X 0,Y 218.33,Z 770.481,A -85,B 0,C 180,E1 -22011.71,E2 -22011.71} C_VEL
LIN {X 0,Y 214.825,Z 782.217,A -85,B 0,C 180,E1 -22013.05,E2 -22013.05} C_VEL
LIN {X 0,Y 211.006,Z 792.966,A -85,B 0,C 180,E1 -22014.641,E2 -22014.641} C_VEL
LIN {X 0,Y 206.902,Z 802.859,A -85,B 0,C 180,E1 -22016.498,E2 -22016.498} C_VEL
LIN {X 0,Y 202.815,Z 811.895,A -85,B 0,C 180,E1 -22018.683,E2 -22018.683} C_VEL
LIN {X 0,Y 198.31,Z 820.804,A -85,B 0,C 180,E1 -22021.418,E2 -22021.418} C_VEL
LIN {X 0,Y 194.42,Z 828.04,A -85,B 0,C 180,E1 -22024.293,E2 -22024.293} C_VEL
LIN {X 0,Y 191.178,Z 833.9,A -85,B 0,C 180,E1 -22027.295,E2 -22027.295} C_VEL
LIN {X 0,Y 188.461,Z 838.601,A -85,B 0,C 180,E1 -22030.39,E2 -22030.39} C_VEL
LIN {X 0,Y 186.168,Z 842.237,A -85,B 0,C 180,E1 -22033.553,E2 -22033.553} C_VEL
LIN {X 0,Y 184.631,Z 844.89,A -85,B 0,C 180,E1 -22036.798,E2 -22036.798} C_VEL
LIN {X 0,Y 183.943,Z 846.169,A -85,B 0,C 180,E1 -22038.987,E2 -22038.987} C_VEL
LIN {X 0,Y 183.28,Z 847.497,A -85,B 0,C 180,E1 -22043.394,E2 -22043.394} C_VEL
LIN {X 0,Y 183.235,Z 847.581,A -85,B 0,C 180,E1 -22045.751,E2 -22045.751} C_VEL
LIN {X 0,Y 183.342,Z 847.281,A -85,B 0,C 180,E1 -22047.803,E2 -22047.803} C_VEL
LIN {X 0,Y 183.496,Z 846.529,A -85,B 0,C 180,E1 -22050,E2 -22050} C_VEL
LIN {X 0,Y 183.378,Z 845.326,A -85,B 0,C 180,E1 -22052.196,E2 -22052.196} C_VEL
LIN {X 0,Y 183.333,Z 843.493,A -85,B 0,C 180,E1 -22054.644,E2 -22054.644} C_VEL
LIN {X 0,Y 183.465,Z 840.336,A -85,B 0,C 180,E1 -22057.705,E2 -22057.705} C_VEL
LIN {X 0,Y 183.982,Z 835.837,A -85,B 0,C 180,E1 -22061.011,E2 -22061.011} C_VEL
LIN {X 0,Y 184.936,Z 830.064,A -85,B 0,C 180,E1 -22064.301,E2 -22064.301} C_VEL
LIN {X 0,Y 186.517,Z 822.78,A -85,B 0,C 180,E1 -22067.544,E2 -22067.544} C_VEL
LIN {X 0,Y 187.978,Z 815.589,A -85,B 0,C 180,E1 -22070.135,E2 -22070.135} C_VEL
LIN {X 0,Y 190.42,Z 805.318,A -85,B 0,C 180,E1 -22073.087,E2 -22073.087} C_VEL
LIN {X 0,Y 192.661,Z 795.178,A -85,B 0,C 180,E1 -22075.379,E2 -22075.379} C_VEL
LIN {X 0,Y 194.63,Z 785.542,A -85,B 0,C 180,E1 -22077.121,E2 -22077.121} C_VEL
LIN {X 0,Y 196.824,Z 773.491,A -85,B 0,C 180,E1 -22078.818,E2 -22078.818} C_VEL
LIN {X 0,Y 198.639,Z 761.07,A -85,B 0,C 180,E1 -22080.129,E2 -22080.129} C_VEL
LIN {X 0,Y 200.031,Z 748.252,A -85,B 0,C 180,E1 -22081.066,E2 -22081.066} C_VEL
LIN {X 0,Y 201.22,Z 728.623,A -85,B 0,C 180,E1 -22081.94,E2 -22081.94} C_VEL
LIN {X 0,Y 202.776,Z 695.599,A -85,B 0,C 180,E1 -22083.264,E2 -22083.264} C_VEL
LIN {X 0,Y 199.652,Z 668.046,A -85,B 0,C 180,E1 -22084.961,E2 -22084.961} C_VEL
LIN {X 0,Y 190.78,Z 643.984,A -85,B 0,C 180,E1 -22087.443,E2 -22087.443} C_VEL
LIN {X 0,Y 187.473,Z 635.771,A -85,B 0,C 180,E1 -22088.434,E2 -22088.434} C_VEL
LIN {X 0,Y 185.555,Z 627.375,A -85,B 0,C 180,E1 -22092.98,E2 -22092.98} C_VEL
LIN {X 0,Y 185.525,Z 627.376,A -85,B 0,C 180,E1 -22097.009,E2 -22097.009} C_VEL
LIN {X 0,Y 185.536,Z 627.374,A -85,B 0,C 180,E1 -22099.912,E2 -22099.912} C_VEL
LIN {X 0,Y 185.559,Z 627.373,A -85,B 0,C 180,E1 -22102.698,E2 -22102.698} C_VEL
LIN {X 0,Y 185.544,Z 627.372,A -85,B 0,C 180,E1 -22107.974,E2 -22107.974} C_VEL
LIN {X 0,Y 185.581,Z 627.367,A -85,B 0,C 180,E1 -22110.574,E2 -22110.574} C_VEL
LIN {X 0,Y 185.578,Z 627.366,A -85,B 0,C 180,E1 -22115.38,E2 -22115.38} C_VEL
LIN {X 0,Y 185.671,Z 627.35,A -85,B 0,C 180,E1 -22121.134,E2 -22121.134} C_VEL
LIN {X 0,Y 185.691,Z 627.354,A -85,B 0,C 180,E1 -22124.636,E2 -22124.636} C_VEL
LIN {X 0,Y 185.921,Z 627.316,A -85,B 0,C 180,E1 -22129.358,E2 -22129.358} C_VEL
LIN {X 0,Y 185.956,Z 627.32,A -85,B 0,C 180,E1 -22133.489,E2 -22133.489} C_VEL
LIN {X 0,Y 186.203,Z 627.286,A -85,B 0,C 180,E1 -22137.836,E2 -22137.836} C_VEL
LIN {X 0,Y 186.405,Z 627.252,A -85,B 0,C 180,E1 -22139.999,E2 -22139.999} C_VEL
LIN {X 0,Y 185.921,Z 627.321,A -85,B 0,C 180,E1 -22144.335,E2 -22144.335} C_VEL
LIN {X 0,Y 186.009,Z 627.312,A -85,B 0,C 180,E1 -22148.691,E2 -22148.691} C_VEL
LIN {X 0,Y 185.728,Z 627.33,A -85,B 0,C 180,E1 -22153.122,E2 -22153.122} C_VEL
LIN {X 0,Y 185.684,Z 627.351,A -85,B 0,C 180,E1 -22157.624,E2 -22157.624} C_VEL
LIN {X 0,Y 185.592,Z 627.359,A -85,B 0,C 180,E1 -22162.251,E2 -22162.251} C_VEL
LIN {X 0,Y 185.555,Z 627.356,A -85,B 0,C 180,E1 -22167.032,E2 -22167.032} C_VEL
LIN {X 0,Y 185.573,Z 627.363,A -85,B 0,C 180,E1 -22169.493,E2 -22169.493} C_VEL
LIN {X 0,Y 185.515,Z 627.369,A -85,B 0,C 180,E1 -22174.627,E2 -22174.627} C_VEL
LIN {X 0,Y 185.563,Z 627.354,A -85,B 0,C 180,E1 -22177.314,E2 -22177.314} C_VEL
LIN {X 0,Y 185.557,Z 627.366,A -85,B 0,C 180,E1 -22180.757,E2 -22180.757} C_VEL
LIN {X 0,Y 185.556,Z 627.37,A -85,B 0,C 180,E1 -22186.022,E2 -22186.022} C_VEL
LIN {X 0,Y 185.505,Z 627.362,A -85,B 0,C 180,E1 -22189.906,E2 -22189.906} C_VEL
LIN {X 0,Y 185.54,Z 627.372,A -85,B 0,C 180,E1 -22192.696,E2 -22192.696} C_VEL
LIN {X 0,Y 185.537,Z 627.368,A -85,B 0,C 180,E1 -22197.975,E2 -22197.975} C_VEL
LIN {X 0,Y 185.577,Z 627.36,A -85,B 0,C 180,E1 -22200.577,E2 -22200.577} C_VEL
LIN {X 0,Y 185.584,Z 627.364,A -85,B 0,C 180,E1 -22205.383,E2 -22205.383} C_VEL
LIN {X 0,Y 185.691,Z 627.354,A -85,B 0,C 180,E1 -22211.116,E2 -22211.116} C_VEL
LIN {X 0,Y 185.725,Z 627.35,A -85,B 0,C 180,E1 -22214.64,E2 -22214.64} C_VEL
LIN {X 0,Y 185.921,Z 627.322,A -85,B 0,C 180,E1 -22219.359,E2 -22219.359} C_VEL
LIN {X 0,Y 185.958,Z 627.318,A -85,B 0,C 180,E1 -22223.49,E2 -22223.49} C_VEL
LIN {X 0,Y 186.206,Z 627.287,A -85,B 0,C 180,E1 -22227.837,E2 -22227.837} C_VEL
LIN {X 0,Y 186.405,Z 627.262,A -85,B 0,C 180,E1 -22230,E2 -22230} C_VEL
LIN {X 0,Y 185.921,Z 627.324,A -85,B 0,C 180,E1 -22234.336,E2 -22234.336} C_VEL
LIN {X 0,Y 185.956,Z 627.322,A -85,B 0,C 180,E1 -22236.851,E2 -22236.851} C_VEL
LIN {X 0,Y 187.024,Z 630.209,A -85,B 0,C 180,E1 -22237.184,E2 -22237.184} C_VEL
LIN {X 0,Y 193.503,Z 643.675,A -85,B 0,C 180,E1 -22238.911,E2 -22238.911} C_VEL
LIN {X 0,Y 201.188,Z 660.992,A -85,B 0,C 180,E1 -22240.856,E2 -22240.856} C_VEL
LIN {X 0,Y 203.887,Z 668.189,A -85,B 0,C 180,E1 -22241.549,E2 -22241.549} C_VEL
LIN {X 0,Y 200.614,Z 727.108,A -85,B 0,C 180,E1 -22243.91,E2 -22243.91} C_VEL
LIN {X 0,Y 199.387,Z 740.86,A -85,B 0,C 180,E1 -22244.871,E2 -22244.871} C_VEL
LIN {X 0,Y 197.812,Z 753.203,A -85,B 0,C 180,E1 -22246.116,E2 -22246.116} C_VEL
LIN {X 0,Y 195.974,Z 765.129,A -85,B 0,C 180,E1 -22247.747,E2 -22247.747} C_VEL
LIN {X 0,Y 193.935,Z 775.678,A -85,B 0,C 180,E1 -22249.577,E2 -22249.577} C_VEL
LIN {X 0,Y 191.638,Z 786.75,A -85,B 0,C 180,E1 -22252.018,E2 -22252.018} C_VEL
LIN {X 0,Y 189.532,Z 796.182,A -85,B 0,C 180,E1 -22254.655,E2 -22254.655} C_VEL
LIN {X 0,Y 187.786,Z 803.817,A -85,B 0,C 180,E1 -22257.287,E2 -22257.287} C_VEL
LIN {X 0,Y 186.16,Z 810.865,A -85,B 0,C 180,E1 -22260.279,E2 -22260.279} C_VEL
LIN {X 0,Y 184.956,Z 816.551,A -85,B 0,C 180,E1 -22263.286,E2 -22263.286} C_VEL
LIN {X 0,Y 183.936,Z 821.568,A -85,B 0,C 180,E1 -22266.643,E2 -22266.643} C_VEL
LIN {X 0,Y 183.269,Z 825.281,A -85,B 0,C 180,E1 -22269.92,E2 -22269.92} C_VEL
LIN {X 0,Y 182.888,Z 828.342,A -85,B 0,C 180,E1 -22273.764,E2 -22273.764} C_VEL
LIN {X 0,Y 182.959,Z 829.856,A -85,B 0,C 180,E1 -22276.872,E2 -22276.872} C_VEL
LIN {X 0,Y 183.425,Z 830.561,A -85,B 0,C 180,E1 -22280.022,E2 -22280.022} C_VEL
LIN {X 0,Y 184.313,Z 830.452,A -85,B 0,C 180,E1 -22283.199,E2 -22283.199} C_VEL
LIN {X 0,Y 185.561,Z 829.485,A -85,B 0,C 180,E1 -22286.43,E2 -22286.43} C_VEL
LIN {X 0,Y 187.291,Z 827.596,A -85,B 0,C 180,E1 -22289.66,E2 -22289.66} C_VEL
LIN {X 0,Y 190.138,Z 823.798,A -85,B 0,C 180,E1 -22293.671,E2 -22293.671} C_VEL
